LIN {X 0,Y 362.033,Z 639.51,A -85,B 0,C 180,E1 -13129.938,E2 -13129.938} C_VEL
LIN {X 0,Y 362.163,Z 639.495,A -85,B 0,C 180,E1 -13133.314,E2 -13133.314} C_VEL
LIN {X 0,Y 362.282,Z 639.48,A -85,B 0,C 180,E1 -13137.777,E2 -13137.777} C_VEL
LIN {X 0,Y 362.428,Z 639.459,A -85,B 0,C 180,E1 -13140,E2 -13140} C_VEL
LIN {X 0,Y 362.282,Z 639.48,A -85,B 0,C 180,E1 -13142.224,E2 -13142.224} C_VEL
LIN {X 0,Y 362.162,Z 639.494,A -85,B 0,C 180,E1 -13146.687,E2 -13146.687} C_VEL
LIN {X 0,Y 362.033,Z 639.507,A -85,B 0,C 180,E1 -13150.062,E2 -13150.062} C_VEL
LIN {X 0,Y 362,Z 639.515,A -85,B 0,C 180,E1 -13153.899,E2 -13153.899} C_VEL
LIN {X 0,Y 361.969,Z 639.52,A -85,B 0,C 180,E1 -13157.939,E2 -13157.939} C_VEL
LIN {X 0,Y 361.863,Z 639.533,A -85,B 0,C 180,E1 -13161.655,E2 -13161.655} C_VEL
LIN {X 0,Y 361.897,Z 639.53,A -85,B 0,C 180,E1 -13165.293,E2 -13165.293} C_VEL
LIN {X 0,Y 361.857,Z 639.512,A -85,B 0,C 180,E1 -13169.074,E2 -13169.074} C_VEL
LIN {X 0,Y 361.851,Z 639.537,A -85,B 0,C 180,E1 -13172.945,E2 -13172.945} C_VEL
LIN {X 0,Y 361.87,Z 639.533,A -85,B 0,C 180,E1 -13175.637,E2 -13175.637} C_VEL
LIN {X 0,Y 361.828,Z 639.538,A -85,B 0,C 180,E1 -13179.019,E2 -13179.019} C_VEL
LIN {X 0,Y 361.835,Z 639.538,A -85,B 0,C 180,E1 -13182.83,E2 -13182.83} C_VEL
LIN {X 0,Y 361.816,Z 639.535,A -85,B 0,C 180,E1 -13185.948,E2 -13185.948} C_VEL
LIN {X 0,Y 361.815,Z 639.547,A -85,B 0,C 180,E1 -13189.249,E2 -13189.249} C_VEL
LIN {X 0,Y 361.865,Z 639.536,A -85,B 0,C 180,E1 -13192.982,E2 -13192.982} C_VEL
LIN {X 0,Y 361.901,Z 639.566,A -85,B 0,C 180,E1 -13195.556,E2 -13195.556} C_VEL
LIN {X 0,Y 363.403,Z 645.852,A -85,B 0,C 180,E1 -13197.377,E2 -13197.377} C_VEL
LIN {X 0,Y 373.289,Z 667.329,A -85,B 0,C 180,E1 -13198.706,E2 -13198.706} C_VEL
LIN {X 0,Y 376.563,Z 675.649,A -85,B 0,C 180,E1 -13199.152,E2 -13199.152} C_VEL
LIN {X 0,Y 374.284,Z 781.835,A -85,B 0,C 180,E1 -13201.238,E2 -13201.238} C_VEL
LIN {X 0,Y 373.515,Z 795.857,A -85,B 0,C 180,E1 -13201.711,E2 -13201.711} C_VEL
LIN {X 0,Y 372.555,Z 809.132,A -85,B 0,C 180,E1 -13202.368,E2 -13202.368} C_VEL
LIN {X 0,Y 371.596,Z 819.142,A -85,B 0,C 180,E1 -13203.005,E2 -13203.005} C_VEL
LIN {X 0,Y 370.352,Z 831.212,A -85,B 0,C 180,E1 -13203.971,E2 -13203.971} C_VEL
LIN {X 0,Y 368.834,Z 843.683,A -85,B 0,C 180,E1 -13205.216,E2 -13205.216} C_VEL
LIN {X 0,Y 367.454,Z 854.256,A -85,B 0,C 180,E1 -13206.521,E2 -13206.521} C_VEL
LIN {X 0,Y 366.023,Z 864.257,A -85,B 0,C 180,E1 -13208.012,E2 -13208.012} C_VEL
LIN {X 0,Y 364.6,Z 873.584,A -85,B 0,C 180,E1 -13209.698,E2 -13209.698} C_VEL
LIN {X 0,Y 363.383,Z 881.912,A -85,B 0,C 180,E1 -13211.543,E2 -13211.543} C_VEL
LIN {X 0,Y 362.532,Z 887.72,A -85,B 0,C 180,E1 -13213.095,E2 -13213.095} C_VEL
LIN {X 0,Y 361.781,Z 892.985,A -85,B 0,C 180,E1 -13214.796,E2 -13214.796} C_VEL
LIN {X 0,Y 361.244,Z 897.486,A -85,B 0,C 180,E1 -13216.596,E2 -13216.596} C_VEL
LIN {X 0,Y 360.734,Z 901.59,A -85,B 0,C 180,E1 -13218.766,E2 -13218.766} C_VEL
LIN {X 0,Y 360.461,Z 904.443,A -85,B 0,C 180,E1 -13221.027,E2 -13221.027} C_VEL
LIN {X 0,Y 360.467,Z 905.926,A -85,B 0,C 180,E1 -13223.282,E2 -13223.282} C_VEL
LIN {X 0,Y 360.37,Z 906.095,A -85,B 0,C 180,E1 -13225.526,E2 -13225.526} C_VEL
LIN {X 0,Y 360.392,Z 904.952,A -85,B 0,C 180,E1 -13227.765,E2 -13227.765} C_VEL
LIN {X 0,Y 360.515,Z 902.485,A -85,B 0,C 180,E1 -13230,E2 -13230} C_VEL
LIN {X 0,Y 360.766,Z 898.613,A -85,B 0,C 180,E1 -13232.233,E2 -13232.233} C_VEL
LIN {X 0,Y 361.422,Z 893.189,A -85,B 0,C 180,E1 -13234.461,E2 -13234.461} C_VEL
LIN {X 0,Y 362.01,Z 888.061,A -85,B 0,C 180,E1 -13236.13,E2 -13236.13} C_VEL
LIN {X 0,Y 362.958,Z 880.664,A -85,B 0,C 180,E1 -13238.07,E2 -13238.07} C_VEL
LIN {X 0,Y 363.669,Z 872.986,A -85,B 0,C 180,E1 -13239.736,E2 -13239.736} C_VEL
LIN {X 0,Y 364.986,Z 863.701,A -85,B 0,C 180,E1 -13241.383,E2 -13241.383} C_VEL
LIN {X 0,Y 366.436,Z 852.377,A -85,B 0,C 180,E1 -13243.024,E2 -13243.024} C_VEL
LIN {X 0,Y 367.722,Z 840.85,A -85,B 0,C 180,E1 -13244.387,E2 -13244.387} C_VEL
LIN {X 0,Y 368.815,Z 829.618,A -85,B 0,C 180,E1 -13245.473,E2 -13245.473} C_VEL
LIN {X 0,Y 369.931,Z 817.471,A -85,B 0,C 180,E1 -13246.415,E2 -13246.415} C_VEL
LIN {X 0,Y 370.111,Z 815.428,A -85,B 0,C 180,E1 -13246.554,E2 -13246.554} C_VEL
LIN {X 0,Y 369.924,Z 810.057,A -85,B 0,C 180,E1 -13246.937,E2 -13246.937} C_VEL
LIN {X 0,Y 367.817,Z 801.278,A -85,B 0,C 180,E1 -13247.579,E2 -13247.579} C_VEL
LIN {X 0,Y 365.572,Z 792.287,A -85,B 0,C 180,E1 -13248.129,E2 -13248.129} C_VEL
LIN {X 0,Y 365.156,Z 786.588,A -85,B 0,C 180,E1 -13248.36,E2 -13248.36} C_VEL
LIN {X 0,Y 365.604,Z 770.654,A -85,B 0,C 180,E1 -13248.747,E2 -13248.747} C_VEL
LIN {X 0,Y 367.59,Z 676.095,A -85,B 0,C 180,E1 -13250.589,E2 -13250.589} C_VEL
LIN {X 0,Y 366.45,Z 671.797,A -85,B 0,C 180,E1 -13250.758,E2 -13250.758} C_VEL
LIN {X 0,Y 359.221,Z 653.429,A -85,B 0,C 180,E1 -13251.672,E2 -13251.672} C_VEL
LIN {X 0,Y 356.012,Z 645.71,A -85,B 0,C 180,E1 -13252.098,E2 -13252.098} C_VEL
LIN {X 0,Y 354.846,Z 640.411,A -85,B 0,C 180,E1 -13253.622,E2 -13253.622} C_VEL
LIN {X 0,Y 354.796,Z 640.417,A -85,B 0,C 180,E1 -13257.104,E2 -13257.104} C_VEL
LIN {X 0,Y 354.796,Z 640.415,A -85,B 0,C 180,E1 -13259.684,E2 -13259.684} C_VEL
LIN {X 0,Y 354.81,Z 640.412,A -85,B 0,C 180,E1 -13263.702,E2 -13263.702} C_VEL
LIN {X 0,Y 354.795,Z 640.414,A -85,B 0,C 180,E1 -13266.46,E2 -13266.46} C_VEL
LIN {X 0,Y 354.771,Z 640.403,A -85,B 0,C 180,E1 -13269.412,E2 -13269.412} C_VEL
LIN {X 0,Y 354.787,Z 640.418,A -85,B 0,C 180,E1 -13272.866,E2 -13272.866} C_VEL
LIN {X 0,Y 354.766,Z 640.416,A -85,B 0,C 180,E1 -13276.103,E2 -13276.103} C_VEL
LIN {X 0,Y 354.767,Z 640.42,A -85,B 0,C 180,E1 -13279.175,E2 -13279.175} C_VEL
LIN {X 0,Y 354.802,Z 640.391,A -85,B 0,C 180,E1 -13282.404,E2 -13282.404} C_VEL
LIN {X 0,Y 354.811,Z 640.403,A -85,B 0,C 180,E1 -13284.94,E2 -13284.94} C_VEL
LIN {X 0,Y 354.796,Z 640.41,A -85,B 0,C 180,E1 -13288.405,E2 -13288.405} C_VEL
LIN {X 0,Y 354.802,Z 640.415,A -85,B 0,C 180,E1 -13291.614,E2 -13291.614} C_VEL
LIN {X 0,Y 354.837,Z 640.397,A -85,B 0,C 180,E1 -13295.657,E2 -13295.657} C_VEL
LIN {X 0,Y 354.829,Z 640.41,A -85,B 0,C 180,E1 -13299.113,E2 -13299.113} C_VEL
LIN {X 0,Y 354.883,Z 640.386,A -85,B 0,C 180,E1 -13302.719,E2 -13302.719} C_VEL
LIN {X 0,Y 354.954,Z 640.393,A -85,B 0,C 180,E1 -13306.255,E2 -13306.255} C_VEL
LIN {X 0,Y 354.959,Z 640.38,A -85,B 0,C 180,E1 -13309.735,E2 -13309.735} C_VEL
LIN {X 0,Y 355.092,Z 640.377,A -85,B 0,C 180,E1 -13313.18,E2 -13313.18} C_VEL
LIN {X 0,Y 355.243,Z 640.36,A -85,B 0,C 180,E1 -13317.732,E2 -13317.732} C_VEL
LIN {X 0,Y 355.376,Z 640.338,A -85,B 0,C 180,E1 -13320,E2 -13320} C_VEL
LIN {X 0,Y 355.245,Z 640.358,A -85,B 0,C 180,E1 -13322.267,E2 -13322.267} C_VEL
LIN {X 0,Y 355.115,Z 640.37,A -85,B 0,C 180,E1 -13326.819,E2 -13326.819} C_VEL
LIN {X 0,Y 355.006,Z 640.386,A -85,B 0,C 180,E1 -13329.112,E2 -13329.112} C_VEL
LIN {X 0,Y 354.924,Z 640.397,A -85,B 0,C 180,E1 -13332.581,E2 -13332.581} C_VEL
LIN {X 0,Y 354.894,Z 640.398,A -85,B 0,C 180,E1 -13336.095,E2 -13336.095} C_VEL
LIN {X 0,Y 354.908,Z 640.396,A -85,B 0,C 180,E1 -13338.471,E2 -13338.471} C_VEL
LIN {X 0,Y 354.817,Z 640.413,A -85,B 0,C 180,E1 -13342.107,E2 -13342.107} C_VEL
LIN {X 0,Y 354.9,Z 640.4,A -85,B 0,C 180,E1 -13345.827,E2 -13345.827} C_VEL
LIN {X 0,Y 354.855,Z 640.406,A -85,B 0,C 180,E1 -13349.678,E2 -13349.678} C_VEL
LIN {X 0,Y 354.807,Z 640.411,A -85,B 0,C 180,E1 -13353.702,E2 -13353.702} C_VEL
LIN {X 0,Y 354.801,Z 640.414,A -85,B 0,C 180,E1 -13356.459,E2 -13356.459} C_VEL
LIN {X 0,Y 354.825,Z 640.406,A -85,B 0,C 180,E1 -13359.423,E2 -13359.423} C_VEL
LIN {X 0,Y 354.806,Z 640.413,A -85,B 0,C 180,E1 -13362.87,E2 -13362.87} C_VEL
LIN {X 0,Y 354.771,Z 640.414,A -85,B 0,C 180,E1 -13366.104,E2 -13366.104} C_VEL
LIN {X 0,Y 354.79,Z 640.415,A -85,B 0,C 180,E1 -13369.179,E2 -13369.179} C_VEL
LIN {X 0,Y 354.813,Z 640.415,A -85,B 0,C 180,E1 -13372.401,E2 -13372.401} C_VEL
LIN {X 0,Y 354.813,Z 640.415,A -85,B 0,C 180,E1 -13374.941,E2 -13374.941} C_VEL
LIN {X 0,Y 354.824,Z 640.498,A -85,B 0,C 180,E1 -13376.358,E2 -13376.358} C_VEL
LIN {X 0,Y 358.492,Z 655.954,A -85,B 0,C 180,E1 -13380.141,E2 -13380.141} C_VEL
LIN {X 0,Y 360.475,Z 665.739,A -85,B 0,C 180,E1 -13382.416,E2 -13382.416} C_VEL
LIN {X 0,Y 360.366,Z 669.663,A -85,B 0,C 180,E1 -13383.251,E2 -13383.251} C_VEL
LIN {X 0,Y 365.528,Z 699.808,A -85,B 0,C 180,E1 -13384.262,E2 -13384.262} C_VEL
LIN {X 0,Y 367.126,Z 709.941,A -85,B 0,C 180,E1 -13384.583,E2 -13384.583} C_VEL
LIN {X 0,Y 365.114,Z 807.088,A -85,B 0,C 180,E1 -13386.496,E2 -13386.496} C_VEL
LIN {X 0,Y 364.378,Z 821.425,A -85,B 0,C 180,E1 -13386.972,E2 -13386.972} C_VEL
LIN {X 0,Y 363.259,Z 835.788,A -85,B 0,C 180,E1 -13387.686,E2 -13387.686} C_VEL
LIN {X 0,Y 362.073,Z 848.948,A -85,B 0,C 180,E1 -13388.574,E2 -13388.574} C_VEL
LIN {X 0,Y 360.801,Z 861.127,A -85,B 0,C 180,E1 -13389.623,E2 -13389.623} C_VEL
LIN {X 0,Y 359.393,Z 872.902,A -85,B 0,C 180,E1 -13390.88,E2 -13390.88} C_VEL
LIN {X 0,Y 358.187,Z 881.703,A -85,B 0,C 180,E1 -13391.999,E2 -13391.999} C_VEL
LIN {X 0,Y 356.842,Z 892.714,A -85,B 0,C 180,E1 -13393.701,E2 -13393.701} C_VEL
LIN {X 0,Y 355.6,Z 902.545,A -85,B 0,C 180,E1 -13395.563,E2 -13395.563} C_VEL
LIN {X 0,Y 354.778,Z 910.501,A -85,B 0,C 180,E1 -13397.414,E2 -13397.414} C_VEL
LIN {X 0,Y 354.09,Z 916.591,A -85,B 0,C 180,E1 -13399.131,E2 -13399.131} C_VEL
LIN {X 0,Y 353.686,Z 921.635,A -85,B 0,C 180,E1 -13400.853,E2 -13400.853} C_VEL
LIN {X 0,Y 353.391,Z 926.828,A -85,B 0,C 180,E1 -13403.147,E2 -13403.147} C_VEL
LIN {X 0,Y 353.329,Z 928.844,A -85,B 0,C 180,E1 -13404.292,E2 -13404.292} C_VEL
LIN {X 0,Y 353.224,Z 931.786,A -85,B 0,C 180,E1 -13406.578,E2 -13406.578} C_VEL
LIN {X 0,Y 353.287,Z 933.347,A -85,B 0,C 180,E1 -13408.86,E2 -13408.86} C_VEL
LIN {X 0,Y 353.328,Z 933.621,A -85,B 0,C 180,E1 -13410,E2 -13410} C_VEL
LIN {X 0,Y 353.199,Z 933.155,A -85,B 0,C 180,E1 -13412.281,E2 -13412.281} C_VEL
LIN {X 0,Y 353.273,Z 931.354,A -85,B 0,C 180,E1 -13414.564,E2 -13414.564} C_VEL
LIN {X 0,Y 353.394,Z 928.176,A -85,B 0,C 180,E1 -13416.853,E2 -13416.853} C_VEL
LIN {X 0,Y 353.707,Z 923.514,A -85,B 0,C 180,E1 -13419.146,E2 -13419.146} C_VEL
LIN {X 0,Y 354.35,Z 917.212,A -85,B 0,C 180,E1 -13421.44,E2 -13421.44} C_VEL
LIN {X 0,Y 355.297,Z 910.221,A -85,B 0,C 180,E1 -13423.44,E2 -13423.44} C_VEL
LIN {X 0,Y 356.34,Z 902.934,A -85,B 0,C 180,E1 -13425.149,E2 -13425.149} C_VEL
LIN {X 0,Y 357.58,Z 894.193,A -85,B 0,C 180,E1 -13426.852,E2 -13426.852} C_VEL
LIN {X 0,Y 359.167,Z 883.624,A -85,B 0,C 180,E1 -13428.54,E2 -13428.54} C_VEL
LIN {X 0,Y 360.968,Z 871.814,A -85,B 0,C 180,E1 -13430.069,E2 -13430.069} C_VEL
LIN {X 0,Y 362.531,Z 860.236,A -85,B 0,C 180,E1 -13431.288,E2 -13431.288} C_VEL
LIN {X 0,Y 364.076,Z 846.936,A -85,B 0,C 180,E1 -13432.411,E2 -13432.411} C_VEL
LIN {X 0,Y 365.535,Z 833.217,A -85,B 0,C 180,E1 -13433.288,E2 -13433.288} C_VEL
LIN {X 0,Y 366.701,Z 819.616,A -85,B 0,C 180,E1 -13433.921,E2 -13433.921} C_VEL
LIN {X 0,Y 367.402,Z 805.854,A -85,B 0,C 180,E1 -13434.36,E2 -13434.36} C_VEL
LIN {X 0,Y 369.645,Z 710.085,A -85,B 0,C 180,E1 -13436.255,E2 -13436.255} C_VEL
LIN {X 0,Y 365.236,Z 685.41,A -85,B 0,C 180,E1 -13437.163,E2 -13437.163} C_VEL
LIN {X 0,Y 361.772,Z 669.821,A -85,B 0,C 180,E1 -13437.814,E2 -13437.814} C_VEL
LIN {X 0,Y 361.611,Z 669.008,A -85,B 0,C 180,E1 -13437.928,E2 -13437.928} C_VEL
LIN {X 0,Y 358.984,Z 656.804,A -85,B 0,C 180,E1 -13440.924,E2 -13440.924} C_VEL
LIN {X 0,Y 355.716,Z 643.633,A -85,B 0,C 180,E1 -13444.366,E2 -13444.366} C_VEL
LIN {X 0,Y 354.851,Z 640.398,A -85,B 0,C 180,E1 -13445.295,E2 -13445.295} C_VEL
LIN {X 0,Y 354.837,Z 640.411,A -85,B 0,C 180,E1 -13449.331,E2 -13449.331} C_VEL
LIN {X 0,Y 354.804,Z 640.411,A -85,B 0,C 180,E1 -13452.87,E2 -13452.87} C_VEL
LIN {X 0,Y 354.776,Z 640.416,A -85,B 0,C 180,E1 -13456.105,E2 -13456.105} C_VEL
LIN {X 0,Y 354.824,Z 640.405,A -85,B 0,C 180,E1 -13459.184,E2 -13459.184} C_VEL
LIN {X 0,Y 354.809,Z 640.395,A -85,B 0,C 180,E1 -13462.402,E2 -13462.402} C_VEL
LIN {X 0,Y 354.813,Z 640.41,A -85,B 0,C 180,E1 -13464.941,E2 -13464.941} C_VEL
LIN {X 0,Y 354.793,Z 640.389,A -85,B 0,C 180,E1 -13468.405,E2 -13468.405} C_VEL
LIN {X 0,Y 354.851,Z 640.407,A -85,B 0,C 180,E1 -13471.619,E2 -13471.619} C_VEL
LIN {X 0,Y 354.9,Z 640.397,A -85,B 0,C 180,E1 -13474.173,E2 -13474.173} C_VEL
LIN {X 0,Y 354.835,Z 640.404,A -85,B 0,C 180,E1 -13477.894,E2 -13477.894} C_VEL
LIN {X 0,Y 354.924,Z 640.392,A -85,B 0,C 180,E1 -13481.891,E2 -13481.891} C_VEL
LIN {X 0,Y 354.944,Z 640.39,A -85,B 0,C 180,E1 -13485.981,E2 -13485.981} C_VEL
LIN {X 0,Y 354.979,Z 640.391,A -85,B 0,C 180,E1 -13489.736,E2 -13489.736} C_VEL
LIN {X 0,Y 355.126,Z 640.372,A -85,B 0,C 180,E1 -13493.181,E2 -13493.181} C_VEL
LIN {X 0,Y 355.245,Z 640.357,A -85,B 0,C 180,E1 -13497.733,E2 -13497.733} C_VEL
LIN {X 0,Y 355.376,Z 640.337,A -85,B 0,C 180,E1 -13500,E2 -13500} C_VEL
LIN {X 0,Y 355.245,Z 640.357,A -85,B 0,C 180,E1 -13502.268,E2 -13502.268} C_VEL
LIN {X 0,Y 355.126,Z 640.373,A -85,B 0,C 180,E1 -13506.82,E2 -13506.82} C_VEL
LIN {X 0,Y 354.979,Z 640.385,A -85,B 0,C 180,E1 -13510.264,E2 -13510.264} C_VEL
LIN {X 0,Y 354.945,Z 640.394,A -85,B 0,C 180,E1 -13514.019,E2 -13514.019} C_VEL
LIN {X 0,Y 354.924,Z 640.398,A -85,B 0,C 180,E1 -13518.109,E2 -13518.109} C_VEL
LIN {X 0,Y 354.817,Z 640.411,A -85,B 0,C 180,E1 -13522.108,E2 -13522.108} C_VEL
LIN {X 0,Y 354.83,Z 640.409,A -85,B 0,C 180,E1 -13525.833,E2 -13525.833} C_VEL
LIN {X 0,Y 354.801,Z 640.392,A -85,B 0,C 180,E1 -13529.684,E2 -13529.684} C_VEL
LIN {X 0,Y 354.789,Z 640.415,A -85,B 0,C 180,E1 -13532.334,E2 -13532.334} C_VEL
LIN {X 0,Y 354.824,Z 640.41,A -85,B 0,C 180,E1 -13535.7,E2 -13535.7} C_VEL
LIN {X 0,Y 354.77,Z 640.412,A -85,B 0,C 180,E1 -13539.413,E2 -13539.413} C_VEL
LIN {X 0,Y 354.787,Z 640.417,A -85,B 0,C 180,E1 -13542.867,E2 -13542.867} C_VEL
LIN {X 0,Y 354.765,Z 640.414,A -85,B 0,C 180,E1 -13546.103,E2 -13546.103} C_VEL
LIN {X 0,Y 354.768,Z 640.425,A -85,B 0,C 180,E1 -13549.176,E2 -13549.176} C_VEL
LIN {X 0,Y 354.802,Z 640.416,A -85,B 0,C 180,E1 -13552.405,E2 -13552.405} C_VEL
LIN {X 0,Y 354.87,Z 640.462,A -85,B 0,C 180,E1 -13555.028,E2 -13555.028} C_VEL
LIN {X 0,Y 356.235,Z 646.109,A -85,B 0,C 180,E1 -13556.718,E2 -13556.718} C_VEL
LIN {X 0,Y 366.574,Z 668.221,A -85,B 0,C 180,E1 -13558.154,E2 -13558.154} C_VEL
LIN {X 0,Y 370.262,Z 677.295,A -85,B 0,C 180,E1 -13558.667,E2 -13558.667} C_VEL
LIN {X 0,Y 367.886,Z 782.415,A -85,B 0,C 180,E1 -13560.769,E2 -13560.769} C_VEL
LIN {X 0,Y 367.076,Z 797.106,A -85,B 0,C 180,E1 -13561.286,E2 -13561.286} C_VEL
LIN {X 0,Y 366.02,Z 810.282,A -85,B 0,C 180,E1 -13561.959,E2 -13561.959} C_VEL
LIN {X 0,Y 365.025,Z 820.541,A -85,B 0,C 180,E1 -13562.634,E2 -13562.634} C_VEL
LIN {X 0,Y 363.539,Z 833.851,A -85,B 0,C 180,E1 -13563.754,E2 -13563.754} C_VEL
LIN {X 0,Y 361.967,Z 845.818,A -85,B 0,C 180,E1 -13565.02,E2 -13565.02} C_VEL
LIN {X 0,Y 360.527,Z 856.284,A -85,B 0,C 180,E1 -13566.379,E2 -13566.379} C_VEL
LIN {X 0,Y 359.094,Z 865.815,A -85,B 0,C 180,E1 -13567.868,E2 -13567.868} C_VEL
LIN {X 0,Y 357.615,Z 874.918,A -85,B 0,C 180,E1 -13569.584,E2 -13569.584} C_VEL
LIN {X 0,Y 356.332,Z 883.589,A -85,B 0,C 180,E1 -13571.605,E2 -13571.605} C_VEL
LIN {X 0,Y 355.347,Z 889.653,A -85,B 0,C 180,E1 -13573.335,E2 -13573.335} C_VEL
LIN {X 0,Y 354.435,Z 896.073,A -85,B 0,C 180,E1 -13575.649,E2 -13575.649} C_VEL
LIN {X 0,Y 353.92,Z 899.781,A -85,B 0,C 180,E1 -13577.383,E2 -13577.383} C_VEL
LIN {X 0,Y 353.476,Z 903.387,A -85,B 0,C 180,E1 -13579.692,E2 -13579.692} C_VEL
LIN {X 0,Y 353.338,Z 905.583,A -85,B 0,C 180,E1 -13581.997,E2 -13581.997} C_VEL
LIN {X 0,Y 353.317,Z 906.405,A -85,B 0,C 180,E1 -13584.035,E2 -13584.035} C_VEL
LIN {X 0,Y 353.28,Z 906.377,A -85,B 0,C 180,E1 -13585.436,E2 -13585.436} C_VEL
LIN {X 0,Y 353.292,Z 905.269,A -85,B 0,C 180,E1 -13587.72,E2 -13587.72} C_VEL
LIN {X 0,Y 353.45,Z 902.837,A -85,B 0,C 180,E1 -13590,E2 -13590} C_VEL
LIN {X 0,Y 353.709,Z 899.017,A -85,B 0,C 180,E1 -13592.278,E2 -13592.278} C_VEL
LIN {X 0,Y 354.386,Z 893.638,A -85,B 0,C 180,E1 -13594.55,E2 -13594.55} C_VEL
LIN {X 0,Y 354.984,Z 888.539,A -85,B 0,C 180,E1 -13596.251,E2 -13596.251} C_VEL
LIN {X 0,Y 355.964,Z 881.204,A -85,B 0,C 180,E1 -13598.23,E2 -13598.23} C_VEL
LIN {X 0,Y 356.705,Z 873.739,A -85,B 0,C 180,E1 -13599.891,E2 -13599.891} C_VEL
LIN {X 0,Y 358.081,Z 864.354,A -85,B 0,C 180,E1 -13601.606,E2 -13601.606} C_VEL
LIN {X 0,Y 359.423,Z 854.174,A -85,B 0,C 180,E1 -13603.139,E2 -13603.139} C_VEL
LIN {X 0,Y 360.757,Z 842.962,A -85,B 0,C 180,E1 -13604.526,E2 -13604.526} C_VEL
LIN {X 0,Y 362.019,Z 830.579,A -85,B 0,C 180,E1 -13605.771,E2 -13605.771} C_VEL
LIN {X 0,Y 363.191,Z 818.604,A -85,B 0,C 180,E1 -13606.729,E2 -13606.729} C_VEL
LIN {X 0,Y 364.218,Z 805.46,A -85,B 0,C 180,E1 -13607.548,E2 -13607.548} C_VEL
LIN {X 0,Y 364.999,Z 791.191,A -85,B 0,C 180,E1 -13608.197,E2 -13608.197} C_VEL
LIN {X 0,Y 365.156,Z 786.588,A -85,B 0,C 180,E1 -13608.36,E2 -13608.36} C_VEL
LIN {X 0,Y 364.747,Z 780.831,A -85,B 0,C 180,E1 -13608.567,E2 -13608.567} C_VEL
LIN {X 0,Y 359.828,Z 762.18,A -85,B 0,C 180,E1 -13609.303,E2 -13609.303} C_VEL
LIN {X 0,Y 359.382,Z 756.37,A -85,B 0,C 180,E1 -13609.454,E2 -13609.454} C_VEL
LIN {X 0,Y 361.125,Z 677.298,A -85,B 0,C 180,E1 -13611.019,E2 -13611.019} C_VEL
LIN {X 0,Y 359.464,Z 672.117,A -85,B 0,C 180,E1 -13611.25,E2 -13611.25} C_VEL
LIN {X 0,Y 352.59,Z 654.789,A -85,B 0,C 180,E1 -13612.144,E2 -13612.144} C_VEL
LIN {X 0,Y 348.833,Z 645.917,A -85,B 0,C 180,E1 -13612.671,E2 -13612.671} C_VEL
LIN {X 0,Y 347.803,Z 641.288,A -85,B 0,C 180,E1 -13614.005,E2 -13614.005} C_VEL
LIN {X 0,Y 347.731,Z 641.298,A -85,B 0,C 180,E1 -13617.701,E2 -13617.701} C_VEL
LIN {X 0,Y 347.732,Z 641.297,A -85,B 0,C 180,E1 -13620.35,E2 -13620.35} C_VEL
LIN {X 0,Y 347.751,Z 641.292,A -85,B 0,C 180,E1 -13624.043,E2 -13624.043} C_VEL
LIN {X 0,Y 347.758,Z 641.292,A -85,B 0,C 180,E1 -13627.322,E2 -13627.322} C_VEL
LIN {X 0,Y 347.744,Z 641.292,A -85,B 0,C 180,E1 -13631.601,E2 -13631.601} C_VEL
LIN {X 0,Y 347.704,Z 641.299,A -85,B 0,C 180,E1 -13635.027,E2 -13635.027} C_VEL
LIN {X 0,Y 347.742,Z 641.291,A -85,B 0,C 180,E1 -13638.399,E2 -13638.399} C_VEL
LIN {X 0,Y 347.758,Z 641.266,A -85,B 0,C 180,E1 -13642.678,E2 -13642.678} C_VEL
LIN {X 0,Y 347.751,Z 641.29,A -85,B 0,C 180,E1 -13645.956,E2 -13645.956} C_VEL
LIN {X 0,Y 347.744,Z 641.282,A -85,B 0,C 180,E1 -13649.651,E2 -13649.651} C_VEL
LIN {X 0,Y 347.751,Z 641.29,A -85,B 0,C 180,E1 -13653.601,E2 -13653.601} C_VEL
LIN {X 0,Y 347.768,Z 641.277,A -85,B 0,C 180,E1 -13656.16,E2 -13656.16} C_VEL
LIN {X 0,Y 347.803,Z 641.283,A -85,B 0,C 180,E1 -13659.908,E2 -13659.908} C_VEL
LIN {X 0,Y 347.835,Z 641.27,A -85,B 0,C 180,E1 -13663.568,E2 -13663.568} C_VEL
LIN {X 0,Y 347.893,Z 641.274,A -85,B 0,C 180,E1 -13667.16,E2 -13667.16} C_VEL
LIN {X 0,Y 347.938,Z 641.257,A -85,B 0,C 180,E1 -13670.7,E2 -13670.7} C_VEL
LIN {X 0,Y 348.046,Z 641.252,A -85,B 0,C 180,E1 -13674.205,E2 -13674.205} C_VEL
LIN {X 0,Y 348.205,Z 641.236,A -85,B 0,C 180,E1 -13677.686,E2 -13677.686} C_VEL
LIN {X 0,Y 348.326,Z 641.216,A -85,B 0,C 180,E1 -13680,E2 -13680} C_VEL
LIN {X 0,Y 348.208,Z 641.234,A -85,B 0,C 180,E1 -13682.313,E2 -13682.313} C_VEL
LIN {X 0,Y 348.083,Z 641.246,A -85,B 0,C 180,E1 -13686.958,E2 -13686.958} C_VEL
LIN {X 0,Y 347.947,Z 641.266,A -85,B 0,C 180,E1 -13689.299,E2 -13689.299} C_VEL
LIN {X 0,Y 347.892,Z 641.272,A -85,B 0,C 180,E1 -13692.839,E2 -13692.839} C_VEL
LIN {X 0,Y 347.843,Z 641.279,A -85,B 0,C 180,E1 -13696.431,E2 -13696.431} C_VEL
LIN {X 0,Y 347.857,Z 641.272,A -85,B 0,C 180,E1 -13698.86,E2 -13698.86} C_VEL
LIN {X 0,Y 347.764,Z 641.286,A -85,B 0,C 180,E1 -13702.58,E2 -13702.58} C_VEL
LIN {X 0,Y 347.812,Z 641.281,A -85,B 0,C 180,E1 -13705.108,E2 -13705.108} C_VEL
LIN {X 0,Y 347.812,Z 641.278,A -85,B 0,C 180,E1 -13707.693,E2 -13707.693} C_VEL
LIN {X 0,Y 347.765,Z 641.289,A -85,B 0,C 180,E1 -13710.346,E2 -13710.346} C_VEL
LIN {X 0,Y 347.746,Z 641.292,A -85,B 0,C 180,E1 -13714.464,E2 -13714.464} C_VEL
LIN {X 0,Y 347.777,Z 641.289,A -85,B 0,C 180,E1 -13717.989,E2 -13717.989} C_VEL
LIN {X 0,Y 347.767,Z 641.288,A -85,B 0,C 180,E1 -13721.828,E2 -13721.828} C_VEL
LIN {X 0,Y 347.768,Z 641.289,A -85,B 0,C 180,E1 -13725.016,E2 -13725.016} C_VEL
LIN {X 0,Y 347.752,Z 641.293,A -85,B 0,C 180,E1 -13728.397,E2 -13728.397} C_VEL
LIN {X 0,Y 347.778,Z 641.289,A -85,B 0,C 180,E1 -13732.01,E2 -13732.01} C_VEL
LIN {X 0,Y 347.745,Z 641.295,A -85,B 0,C 180,E1 -13735.536,E2 -13735.536} C_VEL
LIN {X 0,Y 347.79,Z 641.514,A -85,B 0,C 180,E1 -13735.946,E2 -13735.946} C_VEL
LIN {X 0,Y 350.787,Z 654.007,A -85,B 0,C 180,E1 -13739.1,E2 -13739.1} C_VEL
LIN {X 0,Y 353.5,Z 666.713,A -85,B 0,C 180,E1 -13742.147,E2 -13742.147} C_VEL
LIN {X 0,Y 353.652,Z 669.514,A -85,B 0,C 180,E1 -13742.757,E2 -13742.757} C_VEL
LIN {X 0,Y 358.623,Z 698.233,A -85,B 0,C 180,E1 -13743.746,E2 -13743.746} C_VEL
LIN {X 0,Y 360.601,Z 711.118,A -85,B 0,C 180,E1 -13744.161,E2 -13744.161} C_VEL
LIN {X 0,Y 358.567,Z 805.211,A -85,B 0,C 180,E1 -13746.04,E2 -13746.04} C_VEL
LIN {X 0,Y 357.824,Z 819.341,A -85,B 0,C 180,E1 -13746.487,E2 -13746.487} C_VEL
LIN {X 0,Y 356.792,Z 833.767,A -85,B 0,C 180,E1 -13747.182,E2 -13747.182} C_VEL
LIN {X 0,Y 355.537,Z 847.129,A -85,B 0,C 180,E1 -13748.068,E2 -13748.068} C_VEL
LIN {X 0,Y 354.051,Z 860.472,A -85,B 0,C 180,E1 -13749.217,E2 -13749.217} C_VEL
LIN {X 0,Y 352.63,Z 872.318,A -85,B 0,C 180,E1 -13750.498,E2 -13750.498} C_VEL
LIN {X 0,Y 351.155,Z 883.147,A -85,B 0,C 180,E1 -13751.928,E2 -13751.928} C_VEL
LIN {X 0,Y 349.735,Z 893.871,A -85,B 0,C 180,E1 -13753.66,E2 -13753.66} C_VEL
LIN {X 0,Y 348.583,Z 902.757,A -85,B 0,C 180,E1 -13755.411,E2 -13755.411} C_VEL
LIN {X 0,Y 347.761,Z 910.079,A -85,B 0,C 180,E1 -13757.156,E2 -13757.156} C_VEL
LIN {X 0,Y 347.08,Z 916.2,A -85,B 0,C 180,E1 -13758.909,E2 -13758.909} C_VEL
LIN {X 0,Y 346.524,Z 922.713,A -85,B 0,C 180,E1 -13761.251,E2 -13761.251} C_VEL
LIN {X 0,Y 346.315,Z 926.486,A -85,B 0,C 180,E1 -13763.006,E2 -13763.006} C_VEL
LIN {X 0,Y 346.195,Z 930.173,A -85,B 0,C 180,E1 -13765.342,E2 -13765.342} C_VEL
LIN {X 0,Y 346.125,Z 932.436,A -85,B 0,C 180,E1 -13767.672,E2 -13767.672} C_VEL
LIN {X 0,Y 346.233,Z 933.342,A -85,B 0,C 180,E1 -13770,E2 -13770} C_VEL
LIN {X 0,Y 346.108,Z 932.896,A -85,B 0,C 180,E1 -13772.327,E2 -13772.327} C_VEL
LIN {X 0,Y 346.19,Z 931.116,A -85,B 0,C 180,E1 -13774.658,E2 -13774.658} C_VEL
LIN {X 0,Y 346.319,Z 927.958,A -85,B 0,C 180,E1 -13776.994,E2 -13776.994} C_VEL
LIN {X 0,Y 346.661,Z 923.328,A -85,B 0,C 180,E1 -13779.334,E2 -13779.334} C_VEL
LIN {X 0,Y 347.368,Z 917.054,A -85,B 0,C 180,E1 -13781.673,E2 -13781.673} C_VEL
LIN {X 0,Y 348.359,Z 910.09,A -85,B 0,C 180,E1 -13783.712,E2 -13783.712} C_VEL
LIN {X 0,Y 349.44,Z 902.835,A -85,B 0,C 180,E1 -13785.455,E2 -13785.455} C_VEL
LIN {X 0,Y 350.77,Z 894.13,A -85,B 0,C 180,E1 -13787.189,E2 -13787.189} C_VEL
LIN {X 0,Y 352.427,Z 883.606,A -85,B 0,C 180,E1 -13788.908,E2 -13788.908} C_VEL
LIN {X 0,Y 354.307,Z 871.849,A -85,B 0,C 180,E1 -13790.463,E2 -13790.463} C_VEL
LIN {X 0,Y 356.036,Z 859.28,A -85,B 0,C 180,E1 -13791.809,E2 -13791.809} C_VEL
LIN {X 0,Y 357.524,Z 847.129,A -85,B 0,C 180,E1 -13792.844,E2 -13792.844} C_VEL
LIN {X 0,Y 359.06,Z 833.602,A -85,B 0,C 180,E1 -13793.733,E2 -13793.733} C_VEL
LIN {X 0,Y 360.267,Z 820.297,A -85,B 0,C 180,E1 -13794.375,E2 -13794.375} C_VEL
LIN {X 0,Y 361.051,Z 805.678,A -85,B 0,C 180,E1 -13794.855,E2 -13794.855} C_VEL
LIN {X 0,Y 363.361,Z 710.983,A -85,B 0,C 180,E1 -13796.761,E2 -13796.761} C_VEL
LIN {X 0,Y 358.734,Z 685.235,A -85,B 0,C 180,E1 -13797.74,E2 -13797.74} C_VEL
LIN {X 0,Y 355.938,Z 672.663,A -85,B 0,C 180,E1 -13798.281,E2 -13798.281} C_VEL
LIN {X 0,Y 354.429,Z 668.948,A -85,B 0,C 180,E1 -13798.539,E2 -13798.539} C_VEL
LIN {X 0,Y 352.075,Z 658.15,A -85,B 0,C 180,E1 -13801.265,E2 -13801.265} C_VEL
LIN {X 0,Y 348.935,Z 645.394,A -85,B 0,C 180,E1 -13804.679,E2 -13804.679} C_VEL
LIN {X 0,Y 347.79,Z 641.28,A -85,B 0,C 180,E1 -13805.875,E2 -13805.875} C_VEL
LIN {X 0,Y 347.766,Z 641.289,A -85,B 0,C 180,E1 -13808.791,E2 -13808.791} C_VEL
LIN {X 0,Y 347.766,Z 641.292,A -85,B 0,C 180,E1 -13811.828,E2 -13811.828} C_VEL
LIN {X 0,Y 347.737,Z 641.289,A -85,B 0,C 180,E1 -13815.022,E2 -13815.022} C_VEL
LIN {X 0,Y 347.768,Z 641.279,A -85,B 0,C 180,E1 -13818.394,E2 -13818.394} C_VEL
LIN {X 0,Y 347.777,Z 641.273,A -85,B 0,C 180,E1 -13822.011,E2 -13822.011} C_VEL
LIN {X 0,Y 347.745,Z 641.295,A -85,B 0,C 180,E1 -13825.536,E2 -13825.536} C_VEL
LIN {X 0,Y 347.764,Z 641.27,A -85,B 0,C 180,E1 -13829.654,E2 -13829.654} C_VEL
LIN {X 0,Y 347.852,Z 641.275,A -85,B 0,C 180,E1 -13832.745,E2 -13832.745} C_VEL
LIN {X 0,Y 347.789,Z 641.285,A -85,B 0,C 180,E1 -13836.162,E2 -13836.162} C_VEL
LIN {X 0,Y 347.818,Z 641.286,A -85,B 0,C 180,E1 -13839.91,E2 -13839.91} C_VEL
LIN {X 0,Y 347.868,Z 641.273,A -85,B 0,C 180,E1 -13842.36,E2 -13842.36} C_VEL
LIN {X 0,Y 347.898,Z 641.268,A -85,B 0,C 180,E1 -13845.971,E2 -13845.971} C_VEL
LIN {X 0,Y 347.93,Z 641.269,A -85,B 0,C 180,E1 -13849.526,E2 -13849.526} C_VEL
LIN {X 0,Y 348.092,Z 641.248,A -85,B 0,C 180,E1 -13853.042,E2 -13853.042} C_VEL
LIN {X 0,Y 348.208,Z 641.233,A -85,B 0,C 180,E1 -13857.687,E2 -13857.687} C_VEL
LIN {X 0,Y 348.327,Z 641.215,A -85,B 0,C 180,E1 -13860,E2 -13860} C_VEL
LIN {X 0,Y 348.208,Z 641.234,A -85,B 0,C 180,E1 -13862.314,E2 -13862.314} C_VEL
LIN {X 0,Y 348.092,Z 641.249,A -85,B 0,C 180,E1 -13866.958,E2 -13866.958} C_VEL
LIN {X 0,Y 347.93,Z 641.262,A -85,B 0,C 180,E1 -13870.475,E2 -13870.475} C_VEL
LIN {X 0,Y 347.9,Z 641.271,A -85,B 0,C 180,E1 -13874.15,E2 -13874.15} C_VEL
LIN {X 0,Y 347.893,Z 641.275,A -85,B 0,C 180,E1 -13878.291,E2 -13878.291} C_VEL
LIN {X 0,Y 347.769,Z 641.289,A -85,B 0,C 180,E1 -13881.627,E2 -13881.627} C_VEL
LIN {X 0,Y 347.779,Z 641.291,A -85,B 0,C 180,E1 -13885.111,E2 -13885.111} C_VEL
LIN {X 0,Y 347.743,Z 641.28,A -85,B 0,C 180,E1 -13887.7,E2 -13887.7} C_VEL
LIN {X 0,Y 347.742,Z 641.277,A -85,B 0,C 180,E1 -13890.349,E2 -13890.349} C_VEL
LIN {X 0,Y 347.75,Z 641.286,A -85,B 0,C 180,E1 -13894.044,E2 -13894.044} C_VEL
LIN {X 0,Y 347.759,Z 641.29,A -85,B 0,C 180,E1 -13897.322,E2 -13897.322} C_VEL
LIN {X 0,Y 347.743,Z 641.282,A -85,B 0,C 180,E1 -13901.601,E2 -13901.601} C_VEL
LIN {X 0,Y 347.704,Z 641.29,A -85,B 0,C 180,E1 -13905.028,E2 -13905.028} C_VEL
LIN {X 0,Y 347.743,Z 641.295,A -85,B 0,C 180,E1 -13908.399,E2 -13908.399} C_VEL
LIN {X 0,Y 347.758,Z 641.293,A -85,B 0,C 180,E1 -13912.679,E2 -13912.679} C_VEL
LIN {X 0,Y 347.802,Z 641.418,A -85,B 0,C 180,E1 -13914.483,E2 -13914.483} C_VEL
LIN {X 0,Y 349.139,Z 646.606,A -85,B 0,C 180,E1 -13916.04,E2 -13916.04} C_VEL
LIN {X 0,Y 359.506,Z 668.427,A -85,B 0,C 180,E1 -13917.53,E2 -13917.53} C_VEL
LIN {X 0,Y 363.981,Z 679.086,A -85,B 0,C 180,E1 -13918.167,E2 -13918.167} C_VEL
LIN {X 0,Y 361.584,Z 781.76,A -85,B 0,C 180,E1 -13920.248,E2 -13920.248} C_VEL
LIN {X 0,Y 360.784,Z 796.05,A -85,B 0,C 180,E1 -13920.737,E2 -13920.737} C_VEL
LIN {X 0,Y 359.749,Z 809.186,A -85,B 0,C 180,E1 -13921.399,E2 -13921.399} C_VEL
LIN {X 0,Y 358.627,Z 819.954,A -85,B 0,C 180,E1 -13922.103,E2 -13922.103} C_VEL
LIN {X 0,Y 357.301,Z 831.968,A -85,B 0,C 180,E1 -13923.102,E2 -13923.102} C_VEL
LIN {X 0,Y 355.833,Z 843.105,A -85,B 0,C 180,E1 -13924.245,E2 -13924.245} C_VEL
LIN {X 0,Y 354.155,Z 854.715,A -85,B 0,C 180,E1 -13925.706,E2 -13925.706} C_VEL
LIN {X 0,Y 352.424,Z 865.734,A -85,B 0,C 180,E1 -13927.426,E2 -13927.426} C_VEL
LIN {X 0,Y 350.869,Z 874.896,A -85,B 0,C 180,E1 -13929.174,E2 -13929.174} C_VEL
LIN {X 0,Y 349.465,Z 883.619,A -85,B 0,C 180,E1 -13931.23,E2 -13931.23} C_VEL
LIN {X 0,Y 348.44,Z 889.729,A -85,B 0,C 180,E1 -13932.995,E2 -13932.995} C_VEL
LIN {X 0,Y 347.455,Z 896.191,A -85,B 0,C 180,E1 -13935.355,E2 -13935.355} C_VEL
LIN {X 0,Y 346.765,Z 900.999,A -85,B 0,C 180,E1 -13937.713,E2 -13937.713} C_VEL
LIN {X 0,Y 346.416,Z 903.583,A -85,B 0,C 180,E1 -13939.479,E2 -13939.479} C_VEL
LIN {X 0,Y 346.269,Z 905.813,A -85,B 0,C 180,E1 -13941.832,E2 -13941.832} C_VEL
LIN {X 0,Y 346.245,Z 906.687,A -85,B 0,C 180,E1 -13944.044,E2 -13944.044} C_VEL
LIN {X 0,Y 346.173,Z 906.287,A -85,B 0,C 180,E1 -13946.508,E2 -13946.508} C_VEL
LIN {X 0,Y 346.279,Z 904.555,A -85,B 0,C 180,E1 -13948.837,E2 -13948.837} C_VEL
LIN {X 0,Y 346.476,Z 901.48,A -85,B 0,C 180,E1 -13951.162,E2 -13951.162} C_VEL
LIN {X 0,Y 346.953,Z 896.956,A -85,B 0,C 180,E1 -13953.484,E2 -13953.484} C_VEL
LIN {X 0,Y 347.814,Z 890.792,A -85,B 0,C 180,E1 -13955.799,E2 -13955.799} C_VEL
LIN {X 0,Y 348.38,Z 885.055,A -85,B 0,C 180,E1 -13957.535,E2 -13957.535} C_VEL
LIN {X 0,Y 349.018,Z 880.538,A -85,B 0,C 180,E1 -13958.686,E2 -13958.686} C_VEL
LIN {X 0,Y 349.93,Z 872.718,A -85,B 0,C 180,E1 -13960.414,E2 -13960.414} C_VEL
LIN {X 0,Y 351.438,Z 863.254,A -85,B 0,C 180,E1 -13962.121,E2 -13962.121} C_VEL
LIN {X 0,Y 352.831,Z 852.792,A -85,B 0,C 180,E1 -13963.682,E2 -13963.682} C_VEL
LIN {X 0,Y 354.243,Z 841.234,A -85,B 0,C 180,E1 -13965.094,E2 -13965.094} C_VEL
LIN {X 0,Y 355.456,Z 829.959,A -85,B 0,C 180,E1 -13966.217,E2 -13966.217} C_VEL
LIN {X 0,Y 356.642,Z 817.762,A -85,B 0,C 180,E1 -13967.193,E2 -13967.193} C_VEL
LIN {X 0,Y 357.699,Z 804.274,A -85,B 0,C 180,E1 -13968.026,E2 -13968.026} C_VEL
LIN {X 0,Y 358.432,Z 790.326,A -85,B 0,C 180,E1 -13968.654,E2 -13968.654} C_VEL
LIN {X 0,Y 358.952,Z 775.704,A -85,B 0,C 180,E1 -13969.07,E2 -13969.07} C_VEL
LIN {X 0,Y 359.382,Z 756.37,A -85,B 0,C 180,E1 -13969.454,E2 -13969.454} C_VEL
LIN {X 0,Y 358.925,Z 750.555,A -85,B 0,C 180,E1 -13969.608,E2 -13969.608} C_VEL
LIN {X 0,Y 354.041,Z 731.861,A -85,B 0,C 180,E1 -13970.348,E2 -13970.348} C_VEL
LIN {X 0,Y 353.629,Z 726.045,A -85,B 0,C 180,E1 -13970.504,E2 -13970.504} C_VEL
LIN {X 0,Y 354.658,Z 678.298,A -85,B 0,C 180,E1 -13971.47,E2 -13971.47} C_VEL
LIN {X 0,Y 346.979,Z 658.552,A -85,B 0,C 180,E1 -13972.501,E2 -13972.501} C_VEL
LIN {X 0,Y 341.693,Z 646.317,A -85,B 0,C 180,E1 -13973.212,E2 -13973.212} C_VEL
LIN {X 0,Y 340.738,Z 642.169,A -85,B 0,C 180,E1 -13974.447,E2 -13974.447} C_VEL
LIN {X 0,Y 340.681,Z 642.173,A -85,B 0,C 180,E1 -13978.325,E2 -13978.325} C_VEL
LIN {X 0,Y 340.685,Z 642.174,A -85,B 0,C 180,E1 -13981.046,E2 -13981.046} C_VEL
LIN {X 0,Y 340.718,Z 642.169,A -85,B 0,C 180,E1 -13985.279,E2 -13985.279} C_VEL
LIN {X 0,Y 340.696,Z 642.17,A -85,B 0,C 180,E1 -13988.382,E2 -13988.382} C_VEL
LIN {X 0,Y 340.696,Z 642.169,A -85,B 0,C 180,E1 -13992.044,E2 -13992.044} C_VEL
LIN {X 0,Y 340.652,Z 642.175,A -85,B 0,C 180,E1 -13996.227,E2 -13996.227} C_VEL
LIN {X 0,Y 340.672,Z 642.174,A -85,B 0,C 180,E1 -13998.688,E2 -13998.688} C_VEL
LIN {X 0,Y 340.721,Z 642.148,A -85,B 0,C 180,E1 -14001.77,E2 -14001.77} C_VEL
LIN {X 0,Y 340.725,Z 642.166,A -85,B 0,C 180,E1 -14005.595,E2 -14005.595} C_VEL
LIN {X 0,Y 340.697,Z 642.164,A -85,B 0,C 180,E1 -14008.955,E2 -14008.955} C_VEL
LIN {X 0,Y 340.722,Z 642.169,A -85,B 0,C 180,E1 -14013.012,E2 -14013.012} C_VEL
LIN {X 0,Y 340.743,Z 642.152,A -85,B 0,C 180,E1 -14015.637,E2 -14015.637} C_VEL
LIN {X 0,Y 340.733,Z 642.168,A -85,B 0,C 180,E1 -14019.473,E2 -14019.473} C_VEL
LIN {X 0,Y 340.795,Z 642.142,A -85,B 0,C 180,E1 -14021.98,E2 -14021.98} C_VEL
LIN {X 0,Y 340.872,Z 642.151,A -85,B 0,C 180,E1 -14025.705,E2 -14025.705} C_VEL
LIN {X 0,Y 340.851,Z 642.137,A -85,B 0,C 180,E1 -14029.305,E2 -14029.305} C_VEL
LIN {X 0,Y 341.005,Z 642.13,A -85,B 0,C 180,E1 -14032.896,E2 -14032.896} C_VEL
LIN {X 0,Y 340.833,Z 642.151,A -85,B 0,C 180,E1 -14035.268,E2 -14035.268} C_VEL
LIN {X 0,Y 341.167,Z 642.112,A -85,B 0,C 180,E1 -14037.638,E2 -14037.638} C_VEL
LIN {X 0,Y 341.277,Z 642.093,A -85,B 0,C 180,E1 -14040,E2 -14040} C_VEL
LIN {X 0,Y 341.17,Z 642.111,A -85,B 0,C 180,E1 -14042.361,E2 -14042.361} C_VEL
LIN {X 0,Y 341.053,Z 642.122,A -85,B 0,C 180,E1 -14047.102,E2 -14047.102} C_VEL
LIN {X 0,Y 340.873,Z 642.14,A -85,B 0,C 180,E1 -14050.693,E2 -14050.693} C_VEL
LIN {X 0,Y 340.865,Z 642.145,A -85,B 0,C 180,E1 -14054.324,E2 -14054.324} C_VEL
LIN {X 0,Y 340.84,Z 642.148,A -85,B 0,C 180,E1 -14058.467,E2 -14058.467} C_VEL
LIN {X 0,Y 340.719,Z 642.167,A -85,B 0,C 180,E1 -14061.841,E2 -14061.841} C_VEL
LIN {X 0,Y 340.773,Z 642.159,A -85,B 0,C 180,E1 -14065.664,E2 -14065.664} C_VEL
LIN {X 0,Y 340.742,Z 642.163,A -85,B 0,C 180,E1 -14068.319,E2 -14068.319} C_VEL
LIN {X 0,Y 340.706,Z 642.166,A -85,B 0,C 180,E1 -14071.044,E2 -14071.044} C_VEL
LIN {X 0,Y 340.72,Z 642.167,A -85,B 0,C 180,E1 -14075.278,E2 -14075.278} C_VEL
LIN {X 0,Y 340.719,Z 642.171,A -85,B 0,C 180,E1 -14078.388,E2 -14078.388} C_VEL
LIN {X 0,Y 340.734,Z 642.164,A -85,B 0,C 180,E1 -14082.052,E2 -14082.052} C_VEL
LIN {X 0,Y 340.685,Z 642.17,A -85,B 0,C 180,E1 -14085.461,E2 -14085.461} C_VEL
LIN {X 0,Y 340.687,Z 642.173,A -85,B 0,C 180,E1 -14088.69,E2 -14088.69} C_VEL
LIN {X 0,Y 340.736,Z 642.166,A -85,B 0,C 180,E1 -14091.773,E2 -14091.773} C_VEL
LIN {X 0,Y 340.715,Z 642.297,A -85,B 0,C 180,E1 -14095.458,E2 -14095.458} C_VEL
LIN {X 0,Y 343.608,Z 654.258,A -85,B 0,C 180,E1 -14098.563,E2 -14098.563} C_VEL
LIN {X 0,Y 346.226,Z 666.189,A -85,B 0,C 180,E1 -14101.512,E2 -14101.512} C_VEL
LIN {X 0,Y 346.708,Z 669.139,A -85,B 0,C 180,E1 -14102.21,E2 -14102.21} C_VEL
LIN {X 0,Y 349.029,Z 680.228,A -85,B 0,C 180,E1 -14102.641,E2 -14102.641} C_VEL
LIN {X 0,Y 354.088,Z 711.421,A -85,B 0,C 180,E1 -14103.705,E2 -14103.705} C_VEL
LIN {X 0,Y 352.057,Z 803.315,A -85,B 0,C 180,E1 -14105.568,E2 -14105.568} C_VEL
LIN {X 0,Y 351.304,Z 818.084,A -85,B 0,C 180,E1 -14106.023,E2 -14106.023} C_VEL
LIN {X 0,Y 350.29,Z 831.504,A -85,B 0,C 180,E1 -14106.656,E2 -14106.656} C_VEL
LIN {X 0,Y 349.069,Z 844.74,A -85,B 0,C 180,E1 -14107.509,E2 -14107.509} C_VEL
LIN {X 0,Y 347.574,Z 858.376,A -85,B 0,C 180,E1 -14108.656,E2 -14108.656} C_VEL
LIN {X 0,Y 346.042,Z 870.545,A -85,B 0,C 180,E1 -14109.957,E2 -14109.957} C_VEL
LIN {X 0,Y 344.598,Z 880.637,A -85,B 0,C 180,E1 -14111.263,E2 -14111.263} C_VEL
LIN {X 0,Y 343.096,Z 891.734,A -85,B 0,C 180,E1 -14113.028,E2 -14113.028} C_VEL
LIN {X 0,Y 341.864,Z 900.769,A -85,B 0,C 180,E1 -14114.776,E2 -14114.776} C_VEL
LIN {X 0,Y 340.938,Z 908.528,A -85,B 0,C 180,E1 -14116.591,E2 -14116.591} C_VEL
LIN {X 0,Y 340.056,Z 915.807,A -85,B 0,C 180,E1 -14118.677,E2 -14118.677} C_VEL
LIN {X 0,Y 339.473,Z 922.346,A -85,B 0,C 180,E1 -14121.067,E2 -14121.067} C_VEL
LIN {X 0,Y 339.198,Z 927.223,A -85,B 0,C 180,E1 -14123.456,E2 -14123.456} C_VEL
LIN {X 0,Y 339.097,Z 929.852,A -85,B 0,C 180,E1 -14125.244,E2 -14125.244} C_VEL
LIN {X 0,Y 339.036,Z 932.138,A -85,B 0,C 180,E1 -14127.624,E2 -14127.624} C_VEL
LIN {X 0,Y 339.138,Z 933.064,A -85,B 0,C 180,E1 -14130,E2 -14130} C_VEL
LIN {X 0,Y 339.02,Z 932.639,A -85,B 0,C 180,E1 -14132.376,E2 -14132.376} C_VEL
LIN {X 0,Y 339.093,Z 930.878,A -85,B 0,C 180,E1 -14134.755,E2 -14134.755} C_VEL
LIN {X 0,Y 339.245,Z 927.741,A -85,B 0,C 180,E1 -14137.14,E2 -14137.14} C_VEL
LIN {X 0,Y 339.628,Z 923.142,A -85,B 0,C 180,E1 -14139.529,E2 -14139.529} C_VEL
LIN {X 0,Y 340.393,Z 916.898,A -85,B 0,C 180,E1 -14141.915,E2 -14141.915} C_VEL
LIN {X 0,Y 341.442,Z 909.962,A -85,B 0,C 180,E1 -14143.996,E2 -14143.996} C_VEL
LIN {X 0,Y 342.535,Z 902.738,A -85,B 0,C 180,E1 -14145.775,E2 -14145.775} C_VEL
LIN {X 0,Y 343.968,Z 894.071,A -85,B 0,C 180,E1 -14147.54,E2 -14147.54} C_VEL
LIN {X 0,Y 345.687,Z 883.591,A -85,B 0,C 180,E1 -14149.291,E2 -14149.291} C_VEL
LIN {X 0,Y 347.66,Z 871.888,A -85,B 0,C 180,E1 -14150.873,E2 -14150.873} C_VEL
LIN {X 0,Y 349.26,Z 860.904,A -85,B 0,C 180,E1 -14152.088,E2 -14152.088} C_VEL
LIN {X 0,Y 350.797,Z 849.088,A -85,B 0,C 180,E1 -14153.152,E2 -14153.152} C_VEL
LIN {X 0,Y 352.336,Z 836.198,A -85,B 0,C 180,E1 -14154.058,E2 -14154.058} C_VEL
LIN {X 0,Y 353.659,Z 822.403,A -85,B 0,C 180,E1 -14154.783,E2 -14154.783} C_VEL
LIN {X 0,Y 354.609,Z 808.113,A -85,B 0,C 180,E1 -14155.299,E2 -14155.299} C_VEL
LIN {X 0,Y 356.222,Z 752.31,A -85,B 0,C 180,E1 -14156.454,E2 -14156.454} C_VEL
LIN {X 0,Y 357.09,Z 711.782,A -85,B 0,C 180,E1 -14157.289,E2 -14157.289} C_VEL
LIN {X 0,Y 352.445,Z 686.101,A -85,B 0,C 180,E1 -14158.298,E2 -14158.298} C_VEL
LIN {X 0,Y 350.187,Z 675.675,A -85,B 0,C 180,E1 -14158.755,E2 -14158.755} C_VEL
LIN {X 0,Y 347.222,Z 668.684,A -85,B 0,C 180,E1 -14159.229,E2 -14159.229} C_VEL
LIN {X 0,Y 344.816,Z 658.078,A -85,B 0,C 180,E1 -14162.001,E2 -14162.001} C_VEL
LIN {X 0,Y 341.983,Z 646.745,A -85,B 0,C 180,E1 -14165.129,E2 -14165.129} C_VEL
LIN {X 0,Y 340.71,Z 642.167,A -85,B 0,C 180,E1 -14166.486,E2 -14166.486} C_VEL
LIN {X 0,Y 340.709,Z 642.165,A -85,B 0,C 180,E1 -14169.751,E2 -14169.751} C_VEL
LIN {X 0,Y 340.711,Z 642.165,A -85,B 0,C 180,E1 -14172.899,E2 -14172.899} C_VEL
LIN {X 0,Y 340.711,Z 642.159,A -85,B 0,C 180,E1 -14177.101,E2 -14177.101} C_VEL
LIN {X 0,Y 340.71,Z 642.169,A -85,B 0,C 180,E1 -14180.249,E2 -14180.249} C_VEL
LIN {X 0,Y 340.711,Z 642.154,A -85,B 0,C 180,E1 -14183.559,E2 -14183.559} C_VEL
LIN {X 0,Y 340.694,Z 642.168,A -85,B 0,C 180,E1 -14186.154,E2 -14186.154} C_VEL
LIN {X 0,Y 340.775,Z 642.151,A -85,B 0,C 180,E1 -14190.333,E2 -14190.333} C_VEL
LIN {X 0,Y 340.805,Z 642.153,A -85,B 0,C 180,E1 -14193.02,E2 -14193.02} C_VEL
LIN {X 0,Y 340.729,Z 642.161,A -85,B 0,C 180,E1 -14196.927,E2 -14196.927} C_VEL
LIN {X 0,Y 340.796,Z 642.154,A -85,B 0,C 180,E1 -14200.734,E2 -14200.734} C_VEL
LIN {X 0,Y 340.789,Z 642.156,A -85,B 0,C 180,E1 -14203.219,E2 -14203.219} C_VEL
LIN {X 0,Y 340.845,Z 642.147,A -85,B 0,C 180,E1 -14206.891,E2 -14206.891} C_VEL
LIN {X 0,Y 340.915,Z 642.134,A -85,B 0,C 180,E1 -14210.508,E2 -14210.508} C_VEL
LIN {X 0,Y 341.06,Z 642.125,A -85,B 0,C 180,E1 -14212.898,E2 -14212.898} C_VEL
LIN {X 0,Y 341.169,Z 642.11,A -85,B 0,C 180,E1 -14217.639,E2 -14217.639} C_VEL
LIN {X 0,Y 341.277,Z 642.093,A -85,B 0,C 180,E1 -14220,E2 -14220} C_VEL
LIN {X 0,Y 341.169,Z 642.111,A -85,B 0,C 180,E1 -14222.362,E2 -14222.362} C_VEL
LIN {X 0,Y 341.06,Z 642.125,A -85,B 0,C 180,E1 -14227.102,E2 -14227.102} C_VEL
LIN {X 0,Y 340.872,Z 642.142,A -85,B 0,C 180,E1 -14230.694,E2 -14230.694} C_VEL
LIN {X 0,Y 340.865,Z 642.146,A -85,B 0,C 180,E1 -14234.325,E2 -14234.325} C_VEL
LIN {X 0,Y 340.839,Z 642.151,A -85,B 0,C 180,E1 -14238.467,E2 -14238.467} C_VEL
LIN {X 0,Y 340.719,Z 642.167,A -85,B 0,C 180,E1 -14241.842,E2 -14241.842} C_VEL
LIN {X 0,Y 340.754,Z 642.163,A -85,B 0,C 180,E1 -14244.839,E2 -14244.839} C_VEL
LIN {X 0,Y 340.687,Z 642.15,A -85,B 0,C 180,E1 -14248.325,E2 -14248.325} C_VEL
LIN {X 0,Y 340.696,Z 642.162,A -85,B 0,C 180,E1 -14251.045,E2 -14251.045} C_VEL
LIN {X 0,Y 340.72,Z 642.17,A -85,B 0,C 180,E1 -14255.279,E2 -14255.279} C_VEL
LIN {X 0,Y 340.696,Z 642.171,A -85,B 0,C 180,E1 -14258.383,E2 -14258.383} C_VEL
LIN {X 0,Y 340.695,Z 642.165,A -85,B 0,C 180,E1 -14262.045,E2 -14262.045} C_VEL
LIN {X 0,Y 340.652,Z 642.172,A -85,B 0,C 180,E1 -14266.228,E2 -14266.228} C_VEL
LIN {X 0,Y 340.673,Z 642.177,A -85,B 0,C 180,E1 -14268.689,E2 -14268.689} C_VEL
LIN {X 0,Y 340.721,Z 642.171,A -85,B 0,C 180,E1 -14271.771,E2 -14271.771} C_VEL
LIN {X 0,Y 340.751,Z 642.296,A -85,B 0,C 180,E1 -14273.89,E2 -14273.89} C_VEL
LIN {X 0,Y 341.915,Z 646.786,A -85,B 0,C 180,E1 -14275.306,E2 -14275.306} C_VEL
LIN {X 0,Y 353.037,Z 669.763,A -85,B 0,C 180,E1 -14276.959,E2 -14276.959} C_VEL
LIN {X 0,Y 357.728,Z 680.914,A -85,B 0,C 180,E1 -14277.65,E2 -14277.65} C_VEL
LIN {X 0,Y 355.259,Z 782.434,A -85,B 0,C 180,E1 -14279.746,E2 -14279.746} C_VEL
LIN {X 0,Y 354.417,Z 796.545,A -85,B 0,C 180,E1 -14280.24,E2 -14280.24} C_VEL
LIN {X 0,Y 353.261,Z 810.503,A -85,B 0,C 180,E1 -14280.968,E2 -14280.968} C_VEL
LIN {X 0,Y 352.106,Z 821.351,A -85,B 0,C 180,E1 -14281.703,E2 -14281.703} C_VEL
LIN {X 0,Y 350.509,Z 834.597,A -85,B 0,C 180,E1 -14282.861,E2 -14282.861} C_VEL
LIN {X 0,Y 348.988,Z 845.345,A -85,B 0,C 180,E1 -14284.023,E2 -14284.023} C_VEL
LIN {X 0,Y 347.359,Z 856.076,A -85,B 0,C 180,E1 -14285.44,E2 -14285.44} C_VEL
LIN {X 0,Y 345.79,Z 865.655,A -85,B 0,C 180,E1 -14286.968,E2 -14286.968} C_VEL
LIN {X 0,Y 344.155,Z 874.877,A -85,B 0,C 180,E1 -14288.748,E2 -14288.748} C_VEL
LIN {X 0,Y 342.775,Z 882.717,A -85,B 0,C 180,E1 -14290.589,E2 -14290.589} C_VEL
LIN {X 0,Y 341.569,Z 889.807,A -85,B 0,C 180,E1 -14292.642,E2 -14292.642} C_VEL
LIN {X 0,Y 340.495,Z 896.312,A -85,B 0,C 180,E1 -14295.048,E2 -14295.048} C_VEL
LIN {X 0,Y 339.928,Z 900.098,A -85,B 0,C 180,E1 -14296.855,E2 -14296.855} C_VEL
LIN {X 0,Y 339.361,Z 903.779,A -85,B 0,C 180,E1 -14299.258,E2 -14299.258} C_VEL
LIN {X 0,Y 339.188,Z 906.044,A -85,B 0,C 180,E1 -14301.66,E2 -14301.66} C_VEL
LIN {X 0,Y 339.138,Z 906.969,A -85,B 0,C 180,E1 -14304.053,E2 -14304.053} C_VEL
LIN {X 0,Y 339.096,Z 906.585,A -85,B 0,C 180,E1 -14306.435,E2 -14306.435} C_VEL
LIN {X 0,Y 339.181,Z 904.889,A -85,B 0,C 180,E1 -14308.813,E2 -14308.813} C_VEL
LIN {X 0,Y 339.398,Z 901.849,A -85,B 0,C 180,E1 -14311.187,E2 -14311.187} C_VEL
LIN {X 0,Y 339.89,Z 897.374,A -85,B 0,C 180,E1 -14313.557,E2 -14313.557} C_VEL
LIN {X 0,Y 340.773,Z 891.259,A -85,B 0,C 180,E1 -14315.919,E2 -14315.919} C_VEL
LIN {X 0,Y 341.371,Z 885.559,A -85,B 0,C 180,E1 -14317.69,E2 -14317.69} C_VEL
LIN {X 0,Y 342.015,Z 881.076,A -85,B 0,C 180,E1 -14318.866,E2 -14318.866} C_VEL
LIN {X 0,Y 342.974,Z 873.31,A -85,B 0,C 180,E1 -14320.628,E2 -14320.628} C_VEL
LIN {X 0,Y 344.526,Z 863.91,A -85,B 0,C 180,E1 -14322.368,E2 -14322.368} C_VEL
LIN {X 0,Y 345.992,Z 853.521,A -85,B 0,C 180,E1 -14323.958,E2 -14323.958} C_VEL
LIN {X 0,Y 347.458,Z 842.056,A -85,B 0,C 180,E1 -14325.396,E2 -14325.396} C_VEL
LIN {X 0,Y 348.691,Z 830.907,A -85,B 0,C 180,E1 -14326.541,E2 -14326.541} C_VEL
LIN {X 0,Y 349.919,Z 818.881,A -85,B 0,C 180,E1 -14327.534,E2 -14327.534} C_VEL
LIN {X 0,Y 351.017,Z 805.653,A -85,B 0,C 180,E1 -14328.382,E2 -14328.382} C_VEL
LIN {X 0,Y 351.836,Z 792.14,A -85,B 0,C 180,E1 -14329.017,E2 -14329.017} C_VEL
LIN {X 0,Y 352.355,Z 778.522,A -85,B 0,C 180,E1 -14329.442,E2 -14329.442} C_VEL
LIN {X 0,Y 353.629,Z 726.045,A -85,B 0,C 180,E1 -14330.504,E2 -14330.504} C_VEL
LIN {X 0,Y 353.22,Z 720.237,A -85,B 0,C 180,E1 -14330.66,E2 -14330.66} C_VEL
LIN {X 0,Y 348.351,Z 701.58,A -85,B 0,C 180,E1 -14331.431,E2 -14331.431} C_VEL
LIN {X 0,Y 347.855,Z 695.773,A -85,B 0,C 180,E1 -14331.598,E2 -14331.598} C_VEL
LIN {X 0,Y 348.121,Z 679.783,A -85,B 0,C 180,E1 -14331.934,E2 -14331.934} C_VEL
LIN {X 0,Y 340.985,Z 661.523,A -85,B 0,C 180,E1 -14332.92,E2 -14332.92} C_VEL
LIN {X 0,Y 334.498,Z 646.485,A -85,B 0,C 180,E1 -14333.858,E2 -14333.858} C_VEL
LIN {X 0,Y 333.684,Z 643.048,A -85,B 0,C 180,E1 -14334.913,E2 -14334.913} C_VEL
LIN {X 0,Y 333.648,Z 643.052,A -85,B 0,C 180,E1 -14337.785,E2 -14337.785} C_VEL
LIN {X 0,Y 333.657,Z 643.051,A -85,B 0,C 180,E1 -14340.366,E2 -14340.366} C_VEL
LIN {X 0,Y 333.638,Z 643.053,A -85,B 0,C 180,E1 -14343.209,E2 -14343.209} C_VEL
LIN {X 0,Y 333.676,Z 643.045,A -85,B 0,C 180,E1 -14346.139,E2 -14346.139} C_VEL
LIN {X 0,Y 333.605,Z 643.041,A -85,B 0,C 180,E1 -14349.199,E2 -14349.199} C_VEL
LIN {X 0,Y 333.631,Z 643.051,A -85,B 0,C 180,E1 -14352.499,E2 -14352.499} C_VEL
LIN {X 0,Y 333.596,Z 643.054,A -85,B 0,C 180,E1 -14355.954,E2 -14355.954} C_VEL
LIN {X 0,Y 333.605,Z 643.054,A -85,B 0,C 180,E1 -14359.324,E2 -14359.324} C_VEL
LIN {X 0,Y 333.664,Z 643.021,A -85,B 0,C 180,E1 -14363.168,E2 -14363.168} C_VEL
LIN {X 0,Y 333.675,Z 643.039,A -85,B 0,C 180,E1 -14365.341,E2 -14365.341} C_VEL
LIN {X 0,Y 333.632,Z 643.047,A -85,B 0,C 180,E1 -14368.222,E2 -14368.222} C_VEL
LIN {X 0,Y 333.657,Z 643.04,A -85,B 0,C 180,E1 -14371.022,E2 -14371.022} C_VEL
LIN {X 0,Y 333.698,Z 643.033,A -85,B 0,C 180,E1 -14375.088,E2 -14375.088} C_VEL
LIN {X 0,Y 333.667,Z 643.046,A -85,B 0,C 180,E1 -14379.018,E2 -14379.018} C_VEL
LIN {X 0,Y 333.743,Z 643.023,A -85,B 0,C 180,E1 -14381.586,E2 -14381.586} C_VEL
LIN {X 0,Y 333.811,Z 643.03,A -85,B 0,C 180,E1 -14385.576,E2 -14385.576} C_VEL
LIN {X 0,Y 333.82,Z 643.014,A -85,B 0,C 180,E1 -14389.077,E2 -14389.077} C_VEL
LIN {X 0,Y 333.96,Z 643.008,A -85,B 0,C 180,E1 -14392.746,E2 -14392.746} C_VEL
LIN {X 0,Y 333.797,Z 643.027,A -85,B 0,C 180,E1 -14395.169,E2 -14395.169} C_VEL
LIN {X 0,Y 334.104,Z 642.991,A -85,B 0,C 180,E1 -14397.588,E2 -14397.588} C_VEL
LIN {X 0,Y 334.228,Z 642.971,A -85,B 0,C 180,E1 -14400,E2 -14400} C_VEL
LIN {X 0,Y 334.107,Z 642.991,A -85,B 0,C 180,E1 -14402.411,E2 -14402.411} C_VEL
LIN {X 0,Y 334.009,Z 642.999,A -85,B 0,C 180,E1 -14406.039,E2 -14406.039} C_VEL
LIN {X 0,Y 333.972,Z 643.008,A -85,B 0,C 180,E1 -14408.484,E2 -14408.484} C_VEL
LIN {X 0,Y 333.794,Z 643.03,A -85,B 0,C 180,E1 -14412.154,E2 -14412.154} C_VEL
LIN {X 0,Y 333.781,Z 643.026,A -85,B 0,C 180,E1 -14415.886,E2 -14415.886} C_VEL
LIN {X 0,Y 333.799,Z 643.024,A -85,B 0,C 180,E1 -14418.655,E2 -14418.655} C_VEL
LIN {X 0,Y 333.658,Z 643.046,A -85,B 0,C 180,E1 -14422.28,E2 -14422.28} C_VEL
LIN {X 0,Y 333.737,Z 643.037,A -85,B 0,C 180,E1 -14426.246,E2 -14426.246} C_VEL
LIN {X 0,Y 333.712,Z 643.039,A -85,B 0,C 180,E1 -14428.972,E2 -14428.972} C_VEL
LIN {X 0,Y 333.648,Z 643.05,A -85,B 0,C 180,E1 -14432.588,E2 -14432.588} C_VEL
LIN {X 0,Y 333.678,Z 643.047,A -85,B 0,C 180,E1 -14436.138,E2 -14436.138} C_VEL
LIN {X 0,Y 333.673,Z 643.042,A -85,B 0,C 180,E1 -14439.188,E2 -14439.188} C_VEL
LIN {X 0,Y 333.676,Z 643.046,A -85,B 0,C 180,E1 -14442.508,E2 -14442.508} C_VEL
LIN {X 0,Y 333.622,Z 643.048,A -85,B 0,C 180,E1 -14445.959,E2 -14445.959} C_VEL
LIN {X 0,Y 333.648,Z 643.049,A -85,B 0,C 180,E1 -14449.315,E2 -14449.315} C_VEL
LIN {X 0,Y 333.668,Z 643.048,A -85,B 0,C 180,E1 -14453.167,E2 -14453.167} C_VEL
LIN {X 0,Y 333.695,Z 643.171,A -85,B 0,C 180,E1 -14454.973,E2 -14454.973} C_VEL
LIN {X 0,Y 336.57,Z 655.203,A -85,B 0,C 180,E1 -14458.18,E2 -14458.18} C_VEL
LIN {X 0,Y 339.544,Z 668.773,A -85,B 0,C 180,E1 -14461.607,E2 -14461.607} C_VEL
LIN {X 0,Y 341.322,Z 674.558,A -85,B 0,C 180,E1 -14461.902,E2 -14461.902} C_VEL
LIN {X 0,Y 345.414,Z 698.623,A -85,B 0,C 180,E1 -14462.773,E2 -14462.773} C_VEL
LIN {X 0,Y 347.598,Z 713.262,A -85,B 0,C 180,E1 -14463.267,E2 -14463.267} C_VEL
LIN {X 0,Y 345.458,Z 804.428,A -85,B 0,C 180,E1 -14465.151,E2 -14465.151} C_VEL
LIN {X 0,Y 344.685,Z 818.657,A -85,B 0,C 180,E1 -14465.613,E2 -14465.613} C_VEL
LIN {X 0,Y 343.536,Z 833.127,A -85,B 0,C 180,E1 -14466.329,E2 -14466.329} C_VEL
LIN {X 0,Y 342.258,Z 846.043,A -85,B 0,C 180,E1 -14467.208,E2 -14467.208} C_VEL
LIN {X 0,Y 340.732,Z 859.157,A -85,B 0,C 180,E1 -14468.365,E2 -14468.365} C_VEL
LIN {X 0,Y 339.157,Z 871.137,A -85,B 0,C 180,E1 -14469.69,E2 -14469.69} C_VEL
LIN {X 0,Y 337.518,Z 882.07,A -85,B 0,C 180,E1 -14471.171,E2 -14471.171} C_VEL
LIN {X 0,Y 335.999,Z 892.885,A -85,B 0,C 180,E1 -14472.972,E2 -14472.972} C_VEL
LIN {X 0,Y 334.722,Z 901.951,A -85,B 0,C 180,E1 -14474.816,E2 -14474.816} C_VEL
LIN {X 0,Y 333.802,Z 909.233,A -85,B 0,C 180,E1 -14476.609,E2 -14476.609} C_VEL
LIN {X 0,Y 333.041,Z 915.411,A -85,B 0,C 180,E1 -14478.435,E2 -14478.435} C_VEL
LIN {X 0,Y 332.416,Z 921.977,A -85,B 0,C 180,E1 -14480.876,E2 -14480.876} C_VEL
LIN {X 0,Y 332.115,Z 926.878,A -85,B 0,C 180,E1 -14483.316,E2 -14483.316} C_VEL
LIN {X 0,Y 332.004,Z 929.531,A -85,B 0,C 180,E1 -14485.143,E2 -14485.143} C_VEL
LIN {X 0,Y 331.95,Z 931.839,A -85,B 0,C 180,E1 -14487.573,E2 -14487.573} C_VEL
LIN {X 0,Y 332.043,Z 932.786,A -85,B 0,C 180,E1 -14490,E2 -14490} C_VEL
LIN {X 0,Y 331.936,Z 932.381,A -85,B 0,C 180,E1 -14492.427,E2 -14492.427} C_VEL
LIN {X 0,Y 332.001,Z 930.641,A -85,B 0,C 180,E1 -14494.857,E2 -14494.857} C_VEL
LIN {X 0,Y 332.166,Z 927.525,A -85,B 0,C 180,E1 -14497.293,E2 -14497.293} C_VEL
LIN {X 0,Y 332.566,Z 922.953,A -85,B 0,C 180,E1 -14499.733,E2 -14499.733} C_VEL
LIN {X 0,Y 333.117,Z 918.439,A -85,B 0,C 180,E1 -14501.562,E2 -14501.562} C_VEL
LIN {X 0,Y 334.143,Z 911.957,A -85,B 0,C 180,E1 -14503.687,E2 -14503.687} C_VEL
LIN {X 0,Y 335.288,Z 905.009,A -85,B 0,C 180,E1 -14505.541,E2 -14505.541} C_VEL
LIN {X 0,Y 336.596,Z 897.039,A -85,B 0,C 180,E1 -14507.309,E2 -14507.309} C_VEL
LIN {X 0,Y 338.329,Z 887.269,A -85,B 0,C 180,E1 -14509.097,E2 -14509.097} C_VEL
LIN {X 0,Y 340.239,Z 876.445,A -85,B 0,C 180,E1 -14510.716,E2 -14510.716} C_VEL
LIN {X 0,Y 342.155,Z 864.794,A -85,B 0,C 180,E1 -14512.135,E2 -14512.135} C_VEL
LIN {X 0,Y 343.873,Z 852.7,A -85,B 0,C 180,E1 -14513.327,E2 -14513.327} C_VEL
LIN {X 0,Y 345.513,Z 839.845,A -85,B 0,C 180,E1 -14514.324,E2 -14514.324} C_VEL
LIN {X 0,Y 346.873,Z 826.71,A -85,B 0,C 180,E1 -14515.101,E2 -14515.101} C_VEL
LIN {X 0,Y 348.052,Z 812.478,A -85,B 0,C 180,E1 -14515.69,E2 -14515.69} C_VEL
LIN {X 0,Y 348.732,Z 797.501,A -85,B 0,C 180,E1 -14516.078,E2 -14516.078} C_VEL
LIN {X 0,Y 350.888,Z 712.951,A -85,B 0,C 180,E1 -14517.824,E2 -14517.824} C_VEL
LIN {X 0,Y 346.624,Z 688.896,A -85,B 0,C 180,E1 -14518.79,E2 -14518.79} C_VEL
LIN {X 0,Y 344.371,Z 678.623,A -85,B 0,C 180,E1 -14519.255,E2 -14519.255} C_VEL
LIN {X 0,Y 340.007,Z 668.296,A -85,B 0,C 180,E1 -14519.986,E2 -14519.986} C_VEL
LIN {X 0,Y 336.983,Z 655.513,A -85,B 0,C 180,E1 -14523.465,E2 -14523.465} C_VEL
LIN {X 0,Y 334.402,Z 645.599,A -85,B 0,C 180,E1 -14526.337,E2 -14526.337} C_VEL
LIN {X 0,Y 333.65,Z 643.046,A -85,B 0,C 180,E1 -14527.133,E2 -14527.133} C_VEL
LIN {X 0,Y 333.655,Z 643.04,A -85,B 0,C 180,E1 -14530.766,E2 -14530.766} C_VEL
LIN {X 0,Y 333.618,Z 643.042,A -85,B 0,C 180,E1 -14534.255,E2 -14534.255} C_VEL
LIN {X 0,Y 333.673,Z 643.032,A -85,B 0,C 180,E1 -14537.624,E2 -14537.624} C_VEL
LIN {X 0,Y 333.677,Z 643.039,A -85,B 0,C 180,E1 -14541.197,E2 -14541.197} C_VEL
LIN {X 0,Y 333.686,Z 643.044,A -85,B 0,C 180,E1 -14545.226,E2 -14545.226} C_VEL
LIN {X 0,Y 333.633,Z 643.024,A -85,B 0,C 180,E1 -14548.222,E2 -14548.222} C_VEL
LIN {X 0,Y 333.711,Z 643.036,A -85,B 0,C 180,E1 -14551.028,E2 -14551.028} C_VEL
LIN {X 0,Y 333.736,Z 643.031,A -85,B 0,C 180,E1 -14553.754,E2 -14553.754} C_VEL
LIN {X 0,Y 333.72,Z 643.033,A -85,B 0,C 180,E1 -14557.914,E2 -14557.914} C_VEL
LIN {X 0,Y 333.795,Z 643.024,A -85,B 0,C 180,E1 -14561.59,E2 -14561.59} C_VEL
LIN {X 0,Y 333.809,Z 643.024,A -85,B 0,C 180,E1 -14565.577,E2 -14565.577} C_VEL
LIN {X 0,Y 333.835,Z 643.024,A -85,B 0,C 180,E1 -14569.078,E2 -14569.078} C_VEL
LIN {X 0,Y 334.007,Z 643.004,A -85,B 0,C 180,E1 -14572.747,E2 -14572.747} C_VEL
LIN {X 0,Y 333.81,Z 643.02,A -85,B 0,C 180,E1 -14575.169,E2 -14575.169} C_VEL
LIN {X 0,Y 334.107,Z 642.989,A -85,B 0,C 180,E1 -14577.589,E2 -14577.589} C_VEL
LIN {X 0,Y 334.229,Z 642.97,A -85,B 0,C 180,E1 -14580,E2 -14580} C_VEL
LIN {X 0,Y 334.107,Z 642.991,A -85,B 0,C 180,E1 -14582.412,E2 -14582.412} C_VEL
LIN {X 0,Y 333.993,Z 642.997,A -85,B 0,C 180,E1 -14586.598,E2 -14586.598} C_VEL
LIN {X 0,Y 333.852,Z 643.018,A -85,B 0,C 180,E1 -14589.696,E2 -14589.696} C_VEL
LIN {X 0,Y 333.798,Z 643.028,A -85,B 0,C 180,E1 -14593.392,E2 -14593.392} C_VEL
LIN {X 0,Y 333.749,Z 643.037,A -85,B 0,C 180,E1 -14597.146,E2 -14597.146} C_VEL
LIN {X 0,Y 333.735,Z 643.03,A -85,B 0,C 180,E1 -14599.691,E2 -14599.691} C_VEL
LIN {X 0,Y 333.669,Z 643.038,A -85,B 0,C 180,E1 -14603.591,E2 -14603.591} C_VEL
LIN {X 0,Y 333.665,Z 643.047,A -85,B 0,C 180,E1 -14606.253,E2 -14606.253} C_VEL
LIN {X 0,Y 333.663,Z 643.029,A -85,B 0,C 180,E1 -14610.278,E2 -14610.278} C_VEL
LIN {X 0,Y 333.639,Z 643.047,A -85,B 0,C 180,E1 -14613.209,E2 -14613.209} C_VEL
LIN {X 0,Y 333.677,Z 643.044,A -85,B 0,C 180,E1 -14616.139,E2 -14616.139} C_VEL
LIN {X 0,Y 333.622,Z 643.048,A -85,B 0,C 180,E1 -14619.197,E2 -14619.197} C_VEL
LIN {X 0,Y 333.631,Z 643.05,A -85,B 0,C 180,E1 -14622.5,E2 -14622.5} C_VEL
LIN {X 0,Y 333.596,Z 643.048,A -85,B 0,C 180,E1 -14625.955,E2 -14625.955} C_VEL
LIN {X 0,Y 333.604,Z 643.06,A -85,B 0,C 180,E1 -14629.325,E2 -14629.325} C_VEL
LIN {X 0,Y 333.677,Z 643.132,A -85,B 0,C 180,E1 -14633.248,E2 -14633.248} C_VEL
LIN {X 0,Y 334.767,Z 647.158,A -85,B 0,C 180,E1 -14634.547,E2 -14634.547} C_VEL
LIN {X 0,Y 343.835,Z 665.387,A -85,B 0,C 180,E1 -14635.953,E2 -14635.953} C_VEL
LIN {X 0,Y 351.021,Z 681.586,A -85,B 0,C 180,E1 -14637.041,E2 -14637.041} C_VEL
LIN {X 0,Y 351.589,Z 683.019,A -85,B 0,C 180,E1 -14637.129,E2 -14637.129} C_VEL
LIN {X 0,Y 348.967,Z 783.087,A -85,B 0,C 180,E1 -14639.225,E2 -14639.225} C_VEL
LIN {X 0,Y 348.07,Z 797.555,A -85,B 0,C 180,E1 -14639.752,E2 -14639.752} C_VEL
LIN {X 0,Y 346.779,Z 811.86,A -85,B 0,C 180,E1 -14640.522,E2 -14640.522} C_VEL
LIN {X 0,Y 345.506,Z 823.428,A -85,B 0,C 180,E1 -14641.35,E2 -14641.35} C_VEL
LIN {X 0,Y 343.924,Z 835.696,A -85,B 0,C 180,E1 -14642.462,E2 -14642.462} C_VEL
LIN {X 0,Y 342.12,Z 847.477,A -85,B 0,C 180,E1 -14643.79,E2 -14643.79} C_VEL
LIN {X 0,Y 340.352,Z 858.742,A -85,B 0,C 180,E1 -14645.367,E2 -14645.367} C_VEL
LIN {X 0,Y 338.547,Z 868.848,A -85,B 0,C 180,E1 -14647.093,E2 -14647.093} C_VEL
LIN {X 0,Y 336.906,Z 877.575,A -85,B 0,C 180,E1 -14648.91,E2 -14648.91} C_VEL
LIN {X 0,Y 335.456,Z 885.914,A -85,B 0,C 180,E1 -14651.051,E2 -14651.051} C_VEL
LIN {X 0,Y 334.349,Z 891.695,A -85,B 0,C 180,E1 -14652.886,E2 -14652.886} C_VEL
LIN {X 0,Y 333.54,Z 896.433,A -85,B 0,C 180,E1 -14654.729,E2 -14654.729} C_VEL
LIN {X 0,Y 332.953,Z 900.258,A -85,B 0,C 180,E1 -14656.574,E2 -14656.574} C_VEL
LIN {X 0,Y 332.312,Z 903.976,A -85,B 0,C 180,E1 -14659.028,E2 -14659.028} C_VEL
LIN {X 0,Y 332.123,Z 906.275,A -85,B 0,C 180,E1 -14661.482,E2 -14661.482} C_VEL
LIN {X 0,Y 332.045,Z 907.235,A -85,B 0,C 180,E1 -14663.925,E2 -14663.925} C_VEL
LIN {X 0,Y 332.021,Z 906.884,A -85,B 0,C 180,E1 -14666.359,E2 -14666.359} C_VEL
LIN {X 0,Y 332.083,Z 905.222,A -85,B 0,C 180,E1 -14668.787,E2 -14668.787} C_VEL
LIN {X 0,Y 332.322,Z 902.217,A -85,B 0,C 180,E1 -14671.212,E2 -14671.212} C_VEL
LIN {X 0,Y 332.83,Z 897.784,A -85,B 0,C 180,E1 -14673.632,E2 -14673.632} C_VEL
LIN {X 0,Y 333.459,Z 893.381,A -85,B 0,C 180,E1 -14675.442,E2 -14675.442} C_VEL
LIN {X 0,Y 334.032,Z 888.047,A -85,B 0,C 180,E1 -14677.252,E2 -14677.252} C_VEL
LIN {X 0,Y 335.019,Z 881.612,A -85,B 0,C 180,E1 -14679.052,E2 -14679.052} C_VEL
LIN {X 0,Y 336.046,Z 873.897,A -85,B 0,C 180,E1 -14680.849,E2 -14680.849} C_VEL
LIN {X 0,Y 337.637,Z 864.561,A -85,B 0,C 180,E1 -14682.625,E2 -14682.625} C_VEL
LIN {X 0,Y 339.167,Z 854.246,A -85,B 0,C 180,E1 -14684.245,E2 -14684.245} C_VEL
LIN {X 0,Y 340.684,Z 842.874,A -85,B 0,C 180,E1 -14685.709,E2 -14685.709} C_VEL
LIN {X 0,Y 341.923,Z 831.852,A -85,B 0,C 180,E1 -14686.878,E2 -14686.878} C_VEL
LIN {X 0,Y 343.225,Z 819.991,A -85,B 0,C 180,E1 -14687.887,E2 -14687.887} C_VEL
LIN {X 0,Y 344.363,Z 807.021,A -85,B 0,C 180,E1 -14688.75,E2 -14688.75} C_VEL
LIN {X 0,Y 345.219,Z 793.953,A -85,B 0,C 180,E1 -14689.396,E2 -14689.396} C_VEL
LIN {X 0,Y 345.785,Z 779.844,A -85,B 0,C 180,E1 -14689.865,E2 -14689.865} C_VEL
LIN {X 0,Y 347.855,Z 695.773,A -85,B 0,C 180,E1 -14691.598,E2 -14691.598} C_VEL
LIN {X 0,Y 347.374,Z 691.945,A -85,B 0,C 180,E1 -14691.72,E2 -14691.72} C_VEL
LIN {X 0,Y 346.07,Z 688.356,A -85,B 0,C 180,E1 -14691.902,E2 -14691.902} C_VEL
LIN {X 0,Y 340.044,Z 676.973,A -85,B 0,C 180,E1 -14692.641,E2 -14692.641} C_VEL
LIN {X 0,Y 332.564,Z 658.66,A -85,B 0,C 180,E1 -14693.702,E2 -14693.702} C_VEL
LIN {X 0,Y 327.332,Z 646.911,A -85,B 0,C 180,E1 -14694.459,E2 -14694.459} C_VEL
LIN {X 0,Y 326.606,Z 643.93,A -85,B 0,C 180,E1 -14695.421,E2 -14695.421} C_VEL
LIN {X 0,Y 326.593,Z 643.928,A -85,B 0,C 180,E1 -14698.257,E2 -14698.257} C_VEL
LIN {X 0,Y 326.57,Z 643.933,A -85,B 0,C 180,E1 -14701.098,E2 -14701.098} C_VEL
LIN {X 0,Y 326.609,Z 643.926,A -85,B 0,C 180,E1 -14704.019,E2 -14704.019} C_VEL
LIN {X 0,Y 326.625,Z 643.926,A -85,B 0,C 180,E1 -14707.237,E2 -14707.237} C_VEL
LIN {X 0,Y 326.547,Z 643.926,A -85,B 0,C 180,E1 -14711.124,E2 -14711.124} C_VEL
LIN {X 0,Y 326.562,Z 643.927,A -85,B 0,C 180,E1 -14713.526,E2 -14713.526} C_VEL
LIN {X 0,Y 326.575,Z 643.927,A -85,B 0,C 180,E1 -14717.029,E2 -14717.029} C_VEL
LIN {X 0,Y 326.589,Z 643.918,A -85,B 0,C 180,E1 -14720.778,E2 -14720.778} C_VEL
LIN {X 0,Y 326.613,Z 643.911,A -85,B 0,C 180,E1 -14724.48,E2 -14724.48} C_VEL
LIN {X 0,Y 326.611,Z 643.925,A -85,B 0,C 180,E1 -14727.455,E2 -14727.455} C_VEL
LIN {X 0,Y 326.619,Z 643.913,A -85,B 0,C 180,E1 -14730.336,E2 -14730.336} C_VEL
LIN {X 0,Y 326.644,Z 643.916,A -85,B 0,C 180,E1 -14734.644,E2 -14734.644} C_VEL
LIN {X 0,Y 326.617,Z 643.922,A -85,B 0,C 180,E1 -14738.543,E2 -14738.543} C_VEL
LIN {X 0,Y 326.71,Z 643.905,A -85,B 0,C 180,E1 -14741.175,E2 -14741.175} C_VEL
LIN {X 0,Y 326.766,Z 643.906,A -85,B 0,C 180,E1 -14745.433,E2 -14745.433} C_VEL
LIN {X 0,Y 326.761,Z 643.895,A -85,B 0,C 180,E1 -14748.838,E2 -14748.838} C_VEL
LIN {X 0,Y 326.916,Z 643.885,A -85,B 0,C 180,E1 -14752.589,E2 -14752.589} C_VEL
LIN {X 0,Y 326.765,Z 643.903,A -85,B 0,C 180,E1 -14755.064,E2 -14755.064} C_VEL
LIN {X 0,Y 327.044,Z 643.87,A -85,B 0,C 180,E1 -14757.536,E2 -14757.536} C_VEL
LIN {X 0,Y 327.18,Z 643.849,A -85,B 0,C 180,E1 -14760,E2 -14760} C_VEL
LIN {X 0,Y 327.047,Z 643.87,A -85,B 0,C 180,E1 -14762.463,E2 -14762.463} C_VEL
LIN {X 0,Y 326.984,Z 643.874,A -85,B 0,C 180,E1 -14766.169,E2 -14766.169} C_VEL
LIN {X 0,Y 326.913,Z 643.886,A -85,B 0,C 180,E1 -14768.655,E2 -14768.655} C_VEL
LIN {X 0,Y 326.737,Z 643.909,A -85,B 0,C 180,E1 -14772.421,E2 -14772.421} C_VEL
LIN {X 0,Y 326.756,Z 643.899,A -85,B 0,C 180,E1 -14774.957,E2 -14774.957} C_VEL
LIN {X 0,Y 326.734,Z 643.903,A -85,B 0,C 180,E1 -14778.838,E2 -14778.838} C_VEL
LIN {X 0,Y 326.604,Z 643.92,A -85,B 0,C 180,E1 -14782.788,E2 -14782.788} C_VEL
LIN {X 0,Y 326.691,Z 643.912,A -85,B 0,C 180,E1 -14785.483,E2 -14785.483} C_VEL
LIN {X 0,Y 326.662,Z 643.918,A -85,B 0,C 180,E1 -14789.659,E2 -14789.659} C_VEL
LIN {X 0,Y 326.609,Z 643.924,A -85,B 0,C 180,E1 -14794.019,E2 -14794.019} C_VEL
LIN {X 0,Y 326.631,Z 643.921,A -85,B 0,C 180,E1 -14797.239,E2 -14797.239} C_VEL
LIN {X 0,Y 326.605,Z 643.925,A -85,B 0,C 180,E1 -14800.207,E2 -14800.207} C_VEL
LIN {X 0,Y 326.604,Z 643.924,A -85,B 0,C 180,E1 -14803.518,E2 -14803.518} C_VEL
LIN {X 0,Y 326.583,Z 643.921,A -85,B 0,C 180,E1 -14807.027,E2 -14807.027} C_VEL
LIN {X 0,Y 326.613,Z 643.927,A -85,B 0,C 180,E1 -14810.772,E2 -14810.772} C_VEL
LIN {X 0,Y 326.663,Z 643.95,A -85,B 0,C 180,E1 -14814.439,E2 -14814.439} C_VEL
LIN {X 0,Y 329.566,Z 656.152,A -85,B 0,C 180,E1 -14817.783,E2 -14817.783} C_VEL
LIN {X 0,Y 332.292,Z 668.547,A -85,B 0,C 180,E1 -14821.003,E2 -14821.003} C_VEL
LIN {X 0,Y 335.082,Z 676.361,A -85,B 0,C 180,E1 -14821.427,E2 -14821.427} C_VEL
LIN {X 0,Y 339.86,Z 704.995,A -85,B 0,C 180,E1 -14822.482,E2 -14822.482} C_VEL
LIN {X 0,Y 341.134,Z 713.95,A -85,B 0,C 180,E1 -14822.787,E2 -14822.787} C_VEL
LIN {X 0,Y 338.888,Z 805.526,A -85,B 0,C 180,E1 -14824.717,E2 -14824.717} C_VEL
LIN {X 0,Y 338.018,Z 820.087,A -85,B 0,C 180,E1 -14825.223,E2 -14825.223} C_VEL
LIN {X 0,Y 336.814,Z 834.532,A -85,B 0,C 180,E1 -14825.99,E2 -14825.99} C_VEL
LIN {X 0,Y 335.456,Z 847.29,A -85,B 0,C 180,E1 -14826.902,E2 -14826.902} C_VEL
LIN {X 0,Y 333.9,Z 859.929,A -85,B 0,C 180,E1 -14828.062,E2 -14828.062} C_VEL
LIN {X 0,Y 332.281,Z 871.725,A -85,B 0,C 180,E1 -14829.413,E2 -14829.413} C_VEL
LIN {X 0,Y 330.749,Z 881.528,A -85,B 0,C 180,E1 -14830.77,E2 -14830.77} C_VEL
LIN {X 0,Y 329.148,Z 892.388,A -85,B 0,C 180,E1 -14832.607,E2 -14832.607} C_VEL
LIN {X 0,Y 327.779,Z 901.623,A -85,B 0,C 180,E1 -14834.517,E2 -14834.517} C_VEL
LIN {X 0,Y 326.859,Z 908.808,A -85,B 0,C 180,E1 -14836.319,E2 -14836.319} C_VEL
LIN {X 0,Y 326.038,Z 915.014,A -85,B 0,C 180,E1 -14838.183,E2 -14838.183} C_VEL
LIN {X 0,Y 325.343,Z 921.606,A -85,B 0,C 180,E1 -14840.676,E2 -14840.676} C_VEL
LIN {X 0,Y 325.045,Z 926.533,A -85,B 0,C 180,E1 -14843.17,E2 -14843.17} C_VEL
LIN {X 0,Y 324.915,Z 929.209,A -85,B 0,C 180,E1 -14845.036,E2 -14845.036} C_VEL
LIN {X 0,Y 324.927,Z 930.549,A -85,B 0,C 180,E1 -14846.279,E2 -14846.279} C_VEL
LIN {X 0,Y 324.896,Z 932.192,A -85,B 0,C 180,E1 -14848.76,E2 -14848.76} C_VEL
LIN {X 0,Y 324.948,Z 932.507,A -85,B 0,C 180,E1 -14850,E2 -14850} C_VEL
LIN {X 0,Y 324.854,Z 932.124,A -85,B 0,C 180,E1 -14852.48,E2 -14852.48} C_VEL
LIN {X 0,Y 324.914,Z 930.404,A -85,B 0,C 180,E1 -14854.963,E2 -14854.963} C_VEL
LIN {X 0,Y 325.078,Z 927.31,A -85,B 0,C 180,E1 -14857.453,E2 -14857.453} C_VEL
LIN {X 0,Y 325.517,Z 922.763,A -85,B 0,C 180,E1 -14859.946,E2 -14859.946} C_VEL
LIN {X 0,Y 326.122,Z 918.272,A -85,B 0,C 180,E1 -14861.813,E2 -14861.813} C_VEL
LIN {X 0,Y 327.193,Z 911.818,A -85,B 0,C 180,E1 -14863.984,E2 -14863.984} C_VEL
LIN {X 0,Y 328.344,Z 905.175,A -85,B 0,C 180,E1 -14865.807,E2 -14865.807} C_VEL
LIN {X 0,Y 329.78,Z 896.966,A -85,B 0,C 180,E1 -14867.679,E2 -14867.679} C_VEL
LIN {X 0,Y 331.602,Z 887.238,A -85,B 0,C 180,E1 -14869.5,E2 -14869.5} C_VEL
LIN {X 0,Y 333.6,Z 876.463,A -85,B 0,C 180,E1 -14871.148,E2 -14871.148} C_VEL
LIN {X 0,Y 335.536,Z 865.178,A -85,B 0,C 180,E1 -14872.557,E2 -14872.557} C_VEL
LIN {X 0,Y 337.369,Z 852.86,A -85,B 0,C 180,E1 -14873.804,E2 -14873.804} C_VEL
LIN {X 0,Y 339.079,Z 840.118,A -85,B 0,C 180,E1 -14874.817,E2 -14874.817} C_VEL
LIN {X 0,Y 340.612,Z 825.805,A -85,B 0,C 180,E1 -14875.677,E2 -14875.677} C_VEL
LIN {X 0,Y 341.844,Z 811.193,A -85,B 0,C 180,E1 -14876.274,E2 -14876.274} C_VEL
LIN {X 0,Y 342.558,Z 793.883,A -85,B 0,C 180,E1 -14876.707,E2 -14876.707} C_VEL
LIN {X 0,Y 344.677,Z 713.839,A -85,B 0,C 180,E1 -14878.39,E2 -14878.39} C_VEL
LIN {X 0,Y 340.616,Z 690.749,A -85,B 0,C 180,E1 -14879.342,E2 -14879.342} C_VEL
LIN {X 0,Y 338.569,Z 681.374,A -85,B 0,C 180,E1 -14879.78,E2 -14879.78} C_VEL
LIN {X 0,Y 332.697,Z 667.958,A -85,B 0,C 180,E1 -14880.778,E2 -14880.778} C_VEL
LIN {X 0,Y 329.689,Z 655.109,A -85,B 0,C 180,E1 -14884.395,E2 -14884.395} C_VEL
LIN {X 0,Y 326.615,Z 643.925,A -85,B 0,C 180,E1 -14887.819,E2 -14887.819} C_VEL
LIN {X 0,Y 326.591,Z 643.921,A -85,B 0,C 180,E1 -14891.134,E2 -14891.134} C_VEL
LIN {X 0,Y 326.549,Z 643.926,A -85,B 0,C 180,E1 -14894.747,E2 -14894.747} C_VEL
LIN {X 0,Y 326.598,Z 643.913,A -85,B 0,C 180,E1 -14898.158,E2 -14898.158} C_VEL
LIN {X 0,Y 326.643,Z 643.911,A -85,B 0,C 180,E1 -14901.394,E2 -14901.394} C_VEL
LIN {X 0,Y 326.62,Z 643.922,A -85,B 0,C 180,E1 -14904.851,E2 -14904.851} C_VEL
LIN {X 0,Y 326.61,Z 643.905,A -85,B 0,C 180,E1 -14907.456,E2 -14907.456} C_VEL
LIN {X 0,Y 326.661,Z 643.907,A -85,B 0,C 180,E1 -14910.341,E2 -14910.341} C_VEL
LIN {X 0,Y 326.69,Z 643.912,A -85,B 0,C 180,E1 -14914.517,E2 -14914.517} C_VEL
LIN {X 0,Y 326.647,Z 643.919,A -85,B 0,C 180,E1 -14918.546,E2 -14918.546} C_VEL
LIN {X 0,Y 326.745,Z 643.904,A -85,B 0,C 180,E1 -14921.178,E2 -14921.178} C_VEL
LIN {X 0,Y 326.764,Z 643.903,A -85,B 0,C 180,E1 -14925.433,E2 -14925.433} C_VEL
LIN {X 0,Y 326.771,Z 643.904,A -85,B 0,C 180,E1 -14928.839,E2 -14928.839} C_VEL
LIN {X 0,Y 326.959,Z 643.883,A -85,B 0,C 180,E1 -14932.59,E2 -14932.59} C_VEL
LIN {X 0,Y 326.777,Z 643.896,A -85,B 0,C 180,E1 -14935.065,E2 -14935.065} C_VEL
LIN {X 0,Y 327.047,Z 643.869,A -85,B 0,C 180,E1 -14937.537,E2 -14937.537} C_VEL
LIN {X 0,Y 327.181,Z 643.848,A -85,B 0,C 180,E1 -14940,E2 -14940} C_VEL
LIN {X 0,Y 327.047,Z 643.871,A -85,B 0,C 180,E1 -14942.464,E2 -14942.464} C_VEL
LIN {X 0,Y 326.963,Z 643.872,A -85,B 0,C 180,E1 -14946.589,E2 -14946.589} C_VEL
LIN {X 0,Y 326.807,Z 643.894,A -85,B 0,C 180,E1 -14949.907,E2 -14949.907} C_VEL
LIN {X 0,Y 326.761,Z 643.904,A -85,B 0,C 180,E1 -14953.686,E2 -14953.686} C_VEL
LIN {X 0,Y 326.701,Z 643.913,A -85,B 0,C 180,E1 -14957.528,E2 -14957.528} C_VEL
LIN {X 0,Y 326.661,Z 643.912,A -85,B 0,C 180,E1 -14960.136,E2 -14960.136} C_VEL
LIN {X 0,Y 326.643,Z 643.914,A -85,B 0,C 180,E1 -14964.13,E2 -14964.13} C_VEL
LIN {X 0,Y 326.623,Z 643.901,A -85,B 0,C 180,E1 -14968.254,E2 -14968.254} C_VEL
LIN {X 0,Y 326.575,Z 643.921,A -85,B 0,C 180,E1 -14971.097,E2 -14971.097} C_VEL
LIN {X 0,Y 326.609,Z 643.919,A -85,B 0,C 180,E1 -14974.02,E2 -14974.02} C_VEL
LIN {X 0,Y 326.625,Z 643.921,A -85,B 0,C 180,E1 -14977.238,E2 -14977.238} C_VEL
LIN {X 0,Y 326.545,Z 643.918,A -85,B 0,C 180,E1 -14981.125,E2 -14981.125} C_VEL
LIN {X 0,Y 326.562,Z 643.935,A -85,B 0,C 180,E1 -14983.526,E2 -14983.526} C_VEL
LIN {X 0,Y 326.575,Z 643.934,A -85,B 0,C 180,E1 -14987.029,E2 -14987.029} C_VEL
LIN {X 0,Y 326.584,Z 643.932,A -85,B 0,C 180,E1 -14991.386,E2 -14991.386} C_VEL
LIN {X 0,Y 326.624,Z 644.04,A -85,B 0,C 180,E1 -14992.598,E2 -14992.598} C_VEL
LIN {X 0,Y 327.55,Z 647.5,A -85,B 0,C 180,E1 -14993.738,E2 -14993.738} C_VEL
LIN {X 0,Y 337.145,Z 666.341,A -85,B 0,C 180,E1 -14995.281,E2 -14995.281} C_VEL
LIN {X 0,Y 344.716,Z 683.121,A -85,B 0,C 180,E1 -14996.465,E2 -14996.465} C_VEL
LIN {X 0,Y 345.407,Z 684.921,A -85,B 0,C 180,E1 -14996.576,E2 -14996.576} C_VEL
LIN {X 0,Y 342.759,Z 782.448,A -85,B 0,C 180,E1 -14998.648,E2 -14998.648} C_VEL
LIN {X 0,Y 341.868,Z 796.801,A -85,B 0,C 180,E1 -14999.159,E2 -14999.159} C_VEL
LIN {X 0,Y 340.621,Z 810.601,A -85,B 0,C 180,E1 -14999.892,E2 -14999.892} C_VEL
LIN {X 0,Y 339.311,Z 822.189,A -85,B 0,C 180,E1 -15000.704,E2 -15000.704} C_VEL
LIN {X 0,Y 337.574,Z 835.363,A -85,B 0,C 180,E1 -15001.899,E2 -15001.899} C_VEL
LIN {X 0,Y 335.931,Z 846.072,A -85,B 0,C 180,E1 -15003.101,E2 -15003.101} C_VEL
LIN {X 0,Y 334.23,Z 856.13,A -85,B 0,C 180,E1 -15004.466,E2 -15004.466} C_VEL
LIN {X 0,Y 332.237,Z 867.14,A -85,B 0,C 180,E1 -15006.302,E2 -15006.302} C_VEL
LIN {X 0,Y 330.475,Z 876.203,A -85,B 0,C 180,E1 -15008.151,E2 -15008.151} C_VEL
LIN {X 0,Y 328.804,Z 884.695,A -85,B 0,C 180,E1 -15010.285,E2 -15010.285} C_VEL
LIN {X 0,Y 327.469,Z 891.776,A -85,B 0,C 180,E1 -15012.515,E2 -15012.515} C_VEL
LIN {X 0,Y 326.592,Z 896.556,A -85,B 0,C 180,E1 -15014.396,E2 -15014.396} C_VEL
LIN {X 0,Y 325.979,Z 900.419,A -85,B 0,C 180,E1 -15016.281,E2 -15016.281} C_VEL
LIN {X 0,Y 325.276,Z 904.173,A -85,B 0,C 180,E1 -15018.787,E2 -15018.787} C_VEL
LIN {X 0,Y 325.039,Z 906.507,A -85,B 0,C 180,E1 -15021.295,E2 -15021.295} C_VEL
LIN {X 0,Y 324.958,Z 907.5,A -85,B 0,C 180,E1 -15023.792,E2 -15023.792} C_VEL
LIN {X 0,Y 324.947,Z 907.182,A -85,B 0,C 180,E1 -15026.28,E2 -15026.28} C_VEL
LIN {X 0,Y 324.985,Z 905.555,A -85,B 0,C 180,E1 -15028.761,E2 -15028.761} C_VEL
LIN {X 0,Y 325.232,Z 902.585,A -85,B 0,C 180,E1 -15031.238,E2 -15031.238} C_VEL
LIN {X 0,Y 325.757,Z 898.189,A -85,B 0,C 180,E1 -15033.711,E2 -15033.711} C_VEL
LIN {X 0,Y 326.422,Z 893.825,A -85,B 0,C 180,E1 -15035.56,E2 -15035.56} C_VEL
LIN {X 0,Y 327.015,Z 888.534,A -85,B 0,C 180,E1 -15037.409,E2 -15037.409} C_VEL
LIN {X 0,Y 328.029,Z 882.211,A -85,B 0,C 180,E1 -15039.23,E2 -15039.23} C_VEL
LIN {X 0,Y 329.099,Z 874.475,A -85,B 0,C 180,E1 -15041.081,E2 -15041.081} C_VEL
LIN {X 0,Y 330.762,Z 865.206,A -85,B 0,C 180,E1 -15042.891,E2 -15042.891} C_VEL
LIN {X 0,Y 332.34,Z 854.968,A -85,B 0,C 180,E1 -15044.544,E2 -15044.544} C_VEL
LIN {X 0,Y 333.917,Z 843.688,A -85,B 0,C 180,E1 -15046.036,E2 -15046.036} C_VEL
LIN {X 0,Y 335.184,Z 832.79,A -85,B 0,C 180,E1 -15047.228,E2 -15047.228} C_VEL
LIN {X 0,Y 336.541,Z 821.096,A -85,B 0,C 180,E1 -15048.255,E2 -15048.255} C_VEL
LIN {X 0,Y 337.724,Z 808.383,A -85,B 0,C 180,E1 -15049.133,E2 -15049.133} C_VEL
LIN {X 0,Y 338.642,Z 794.855,A -85,B 0,C 180,E1 -15049.828,E2 -15049.828} C_VEL
LIN {X 0,Y 339.264,Z 781.137,A -85,B 0,C 180,E1 -15050.303,E2 -15050.303} C_VEL
LIN {X 0,Y 341.804,Z 681.724,A -85,B 0,C 180,E1 -15052.389,E2 -15052.389} C_VEL
LIN {X 0,Y 340.044,Z 676.973,A -85,B 0,C 180,E1 -15052.641,E2 -15052.641} C_VEL
LIN {X 0,Y 337.46,Z 672.038,A -85,B 0,C 180,E1 -15052.969,E2 -15052.969} C_VEL
LIN {X 0,Y 324.785,Z 656.442,A -85,B 0,C 180,E1 -15054.456,E2 -15054.456} C_VEL
LIN {X 0,Y 322.891,Z 653.26,A -85,B 0,C 180,E1 -15054.71,E2 -15054.71} C_VEL
LIN {X 0,Y 320.151,Z 647.162,A -85,B 0,C 180,E1 -15055.137,E2 -15055.137} C_VEL
LIN {X 0,Y 319.538,Z 644.807,A -85,B 0,C 180,E1 -15055.944,E2 -15055.944} C_VEL
LIN {X 0,Y 319.527,Z 644.805,A -85,B 0,C 180,E1 -15058.94,E2 -15058.94} C_VEL
LIN {X 0,Y 319.523,Z 644.81,A -85,B 0,C 180,E1 -15061.863,E2 -15061.863} C_VEL
LIN {X 0,Y 319.581,Z 644.801,A -85,B 0,C 180,E1 -15065.542,E2 -15065.542} C_VEL
LIN {X 0,Y 319.531,Z 644.79,A -85,B 0,C 180,E1 -15069.662,E2 -15069.662} C_VEL
LIN {X 0,Y 319.522,Z 644.804,A -85,B 0,C 180,E1 -15073.46,E2 -15073.46} C_VEL
LIN {X 0,Y 319.553,Z 644.802,A -85,B 0,C 180,E1 -15077.016,E2 -15077.016} C_VEL
LIN {X 0,Y 319.548,Z 644.802,A -85,B 0,C 180,E1 -15080.37,E2 -15080.37} C_VEL
LIN {X 0,Y 319.581,Z 644.787,A -85,B 0,C 180,E1 -15084.457,E2 -15084.457} C_VEL
LIN {X 0,Y 319.527,Z 644.804,A -85,B 0,C 180,E1 -15088.137,E2 -15088.137} C_VEL
LIN {X 0,Y 319.574,Z 644.801,A -85,B 0,C 180,E1 -15091.603,E2 -15091.603} C_VEL
LIN {X 0,Y 319.575,Z 644.79,A -85,B 0,C 180,E1 -15095.301,E2 -15095.301} C_VEL
LIN {X 0,Y 319.568,Z 644.801,A -85,B 0,C 180,E1 -15098.045,E2 -15098.045} C_VEL
LIN {X 0,Y 319.627,Z 644.777,A -85,B 0,C 180,E1 -15102.071,E2 -15102.071} C_VEL
LIN {X 0,Y 319.735,Z 644.781,A -85,B 0,C 180,E1 -15106.007,E2 -15106.007} C_VEL
LIN {X 0,Y 319.738,Z 644.765,A -85,B 0,C 180,E1 -15109.872,E2 -15109.872} C_VEL
LIN {X 0,Y 319.904,Z 644.763,A -85,B 0,C 180,E1 -15113.693,E2 -15113.693} C_VEL
LIN {X 0,Y 319.988,Z 644.748,A -85,B 0,C 180,E1 -15117.482,E2 -15117.482} C_VEL
LIN {X 0,Y 320.132,Z 644.727,A -85,B 0,C 180,E1 -15120,E2 -15120} C_VEL
LIN {X 0,Y 319.991,Z 644.749,A -85,B 0,C 180,E1 -15122.517,E2 -15122.517} C_VEL
LIN {X 0,Y 319.94,Z 644.751,A -85,B 0,C 180,E1 -15126.305,E2 -15126.305} C_VEL
LIN {X 0,Y 319.84,Z 644.767,A -85,B 0,C 180,E1 -15128.848,E2 -15128.848} C_VEL
LIN {X 0,Y 319.684,Z 644.786,A -85,B 0,C 180,E1 -15132.699,E2 -15132.699} C_VEL
LIN {X 0,Y 319.702,Z 644.778,A -85,B 0,C 180,E1 -15135.295,E2 -15135.295} C_VEL
LIN {X 0,Y 319.675,Z 644.782,A -85,B 0,C 180,E1 -15139.255,E2 -15139.255} C_VEL
LIN {X 0,Y 319.562,Z 644.797,A -85,B 0,C 180,E1 -15143.32,E2 -15143.32} C_VEL
LIN {X 0,Y 319.636,Z 644.795,A -85,B 0,C 180,E1 -15146.088,E2 -15146.088} C_VEL
LIN {X 0,Y 319.591,Z 644.799,A -85,B 0,C 180,E1 -15148.933,E2 -15148.933} C_VEL
LIN {X 0,Y 319.535,Z 644.804,A -85,B 0,C 180,E1 -15151.861,E2 -15151.861} C_VEL
LIN {X 0,Y 319.581,Z 644.801,A -85,B 0,C 180,E1 -15155.543,E2 -15155.543} C_VEL
LIN {X 0,Y 319.599,Z 644.799,A -85,B 0,C 180,E1 -15158.004,E2 -15158.004} C_VEL
LIN {X 0,Y 319.573,Z 644.8,A -85,B 0,C 180,E1 -15161.606,E2 -15161.606} C_VEL
LIN {X 0,Y 319.523,Z 644.806,A -85,B 0,C 180,E1 -15165.263,E2 -15165.263} C_VEL
LIN {X 0,Y 319.53,Z 644.808,A -85,B 0,C 180,E1 -15168.712,E2 -15168.712} C_VEL
LIN {X 0,Y 319.579,Z 644.804,A -85,B 0,C 180,E1 -15172.344,E2 -15172.344} C_VEL
LIN {X 0,Y 319.618,Z 644.97,A -85,B 0,C 180,E1 -15173.946,E2 -15173.946} C_VEL
LIN {X 0,Y 322.455,Z 656.813,A -85,B 0,C 180,E1 -15177.288,E2 -15177.288} C_VEL
LIN {X 0,Y 325.044,Z 668.351,A -85,B 0,C 180,E1 -15180.354,E2 -15180.354} C_VEL
LIN {X 0,Y 328.931,Z 678.63,A -85,B 0,C 180,E1 -15180.95,E2 -15180.95} C_VEL
LIN {X 0,Y 333.394,Z 705.711,A -85,B 0,C 180,E1 -15181.973,E2 -15181.973} C_VEL
LIN {X 0,Y 334.699,Z 714.937,A -85,B 0,C 180,E1 -15182.296,E2 -15182.296} C_VEL
LIN {X 0,Y 332.399,Z 805.086,A -85,B 0,C 180,E1 -15184.23,E2 -15184.23} C_VEL
LIN {X 0,Y 331.505,Z 819.726,A -85,B 0,C 180,E1 -15184.744,E2 -15184.744} C_VEL
LIN {X 0,Y 330.295,Z 833.626,A -85,B 0,C 180,E1 -15185.485,E2 -15185.485} C_VEL
LIN {X 0,Y 328.898,Z 846.524,A -85,B 0,C 180,E1 -15186.414,E2 -15186.414} C_VEL
LIN {X 0,Y 327.232,Z 859.56,A -85,B 0,C 180,E1 -15187.626,E2 -15187.626} C_VEL
LIN {X 0,Y 325.412,Z 872.31,A -85,B 0,C 180,E1 -15189.123,E2 -15189.123} C_VEL
LIN {X 0,Y 323.679,Z 882.954,A -85,B 0,C 180,E1 -15190.663,E2 -15190.663} C_VEL
LIN {X 0,Y 322.057,Z 893.533,A -85,B 0,C 180,E1 -15192.539,E2 -15192.539} C_VEL
LIN {X 0,Y 320.698,Z 902.257,A -85,B 0,C 180,E1 -15194.427,E2 -15194.427} C_VEL
LIN {X 0,Y 319.721,Z 909.508,A -85,B 0,C 180,E1 -15196.331,E2 -15196.331} C_VEL
LIN {X 0,Y 318.763,Z 916.447,A -85,B 0,C 180,E1 -15198.555,E2 -15198.555} C_VEL
LIN {X 0,Y 318.286,Z 921.234,A -85,B 0,C 180,E1 -15200.467,E2 -15200.467} C_VEL
LIN {X 0,Y 317.97,Z 926.188,A -85,B 0,C 180,E1 -15203.017,E2 -15203.017} C_VEL
LIN {X 0,Y 317.832,Z 928.886,A -85,B 0,C 180,E1 -15204.925,E2 -15204.925} C_VEL
LIN {X 0,Y 317.788,Z 931.24,A -85,B 0,C 180,E1 -15207.465,E2 -15207.465} C_VEL
LIN {X 0,Y 317.853,Z 932.229,A -85,B 0,C 180,E1 -15210,E2 -15210} C_VEL
LIN {X 0,Y 317.774,Z 931.867,A -85,B 0,C 180,E1 -15212.535,E2 -15212.535} C_VEL
LIN {X 0,Y 317.833,Z 930.168,A -85,B 0,C 180,E1 -15215.074,E2 -15215.074} C_VEL
LIN {X 0,Y 318.004,Z 927.095,A -85,B 0,C 180,E1 -15217.62,E2 -15217.62} C_VEL
LIN {X 0,Y 318.486,Z 922.573,A -85,B 0,C 180,E1 -15220.168,E2 -15220.168} C_VEL
LIN {X 0,Y 319.135,Z 918.107,A -85,B 0,C 180,E1 -15222.076,E2 -15222.076} C_VEL
LIN {X 0,Y 320.275,Z 911.681,A -85,B 0,C 180,E1 -15224.292,E2 -15224.292} C_VEL
LIN {X 0,Y 321.688,Z 903.715,A -85,B 0,C 180,E1 -15226.5,E2 -15226.5} C_VEL
LIN {X 0,Y 323.299,Z 895.408,A -85,B 0,C 180,E1 -15228.373,E2 -15228.373} C_VEL
LIN {X 0,Y 325.197,Z 885.426,A -85,B 0,C 180,E1 -15230.23,E2 -15230.23} C_VEL
LIN {X 0,Y 327.421,Z 874.345,A -85,B 0,C 180,E1 -15231.898,E2 -15231.898} C_VEL
LIN {X 0,Y 329.321,Z 863.253,A -85,B 0,C 180,E1 -15233.266,E2 -15233.266} C_VEL
LIN {X 0,Y 331.336,Z 849.724,A -85,B 0,C 180,E1 -15234.599,E2 -15234.599} C_VEL
LIN {X 0,Y 333.199,Z 836.117,A -85,B 0,C 180,E1 -15235.62,E2 -15235.62} C_VEL
LIN {X 0,Y 334.657,Z 822.585,A -85,B 0,C 180,E1 -15236.378,E2 -15236.378} C_VEL
LIN {X 0,Y 335.751,Z 808.791,A -85,B 0,C 180,E1 -15236.914,E2 -15236.914} C_VEL
LIN {X 0,Y 336.57,Z 786.51,A -85,B 0,C 180,E1 -15237.437,E2 -15237.437} C_VEL
LIN {X 0,Y 338.535,Z 714.812,A -85,B 0,C 180,E1 -15238.971,E2 -15238.971} C_VEL
LIN {X 0,Y 334.454,Z 691.62,A -85,B 0,C 180,E1 -15239.959,E2 -15239.959} C_VEL
LIN {X 0,Y 332.789,Z 684.088,A -85,B 0,C 180,E1 -15240.325,E2 -15240.325} C_VEL
LIN {X 0,Y 326.815,Z 670.892,A -85,B 0,C 180,E1 -15241.323,E2 -15241.323} C_VEL
LIN {X 0,Y 325.418,Z 667.617,A -85,B 0,C 180,E1 -15241.61,E2 -15241.61} C_VEL
LIN {X 0,Y 322.812,Z 656.455,A -85,B 0,C 180,E1 -15244.854,E2 -15244.854} C_VEL
LIN {X 0,Y 319.615,Z 644.796,A -85,B 0,C 180,E1 -15248.554,E2 -15248.554} C_VEL
LIN {X 0,Y 319.578,Z 644.795,A -85,B 0,C 180,E1 -15252.979,E2 -15252.979} C_VEL
LIN {X 0,Y 319.578,Z 644.791,A -85,B 0,C 180,E1 -15257.021,E2 -15257.021} C_VEL
LIN {X 0,Y 319.581,Z 644.801,A -85,B 0,C 180,E1 -15260.376,E2 -15260.376} C_VEL
LIN {X 0,Y 319.56,Z 644.787,A -85,B 0,C 180,E1 -15263.573,E2 -15263.573} C_VEL
LIN {X 0,Y 319.577,Z 644.795,A -85,B 0,C 180,E1 -15266.687,E2 -15266.687} C_VEL
LIN {X 0,Y 319.591,Z 644.776,A -85,B 0,C 180,E1 -15269.617,E2 -15269.617} C_VEL
LIN {X 0,Y 319.609,Z 644.794,A -85,B 0,C 180,E1 -15272.498,E2 -15272.498} C_VEL
LIN {X 0,Y 319.605,Z 644.795,A -85,B 0,C 180,E1 -15275.304,E2 -15275.304} C_VEL
LIN {X 0,Y 319.597,Z 644.792,A -85,B 0,C 180,E1 -15278.048,E2 -15278.048} C_VEL
LIN {X 0,Y 319.69,Z 644.782,A -85,B 0,C 180,E1 -15280.962,E2 -15280.962} C_VEL
LIN {X 0,Y 319.732,Z 644.779,A -85,B 0,C 180,E1 -15285.276,E2 -15285.276} C_VEL
LIN {X 0,Y 319.754,Z 644.775,A -85,B 0,C 180,E1 -15289.873,E2 -15289.873} C_VEL
LIN {X 0,Y 319.913,Z 644.759,A -85,B 0,C 180,E1 -15292.426,E2 -15292.426} C_VEL
LIN {X 0,Y 319.746,Z 644.772,A -85,B 0,C 180,E1 -15294.956,E2 -15294.956} C_VEL
LIN {X 0,Y 319.991,Z 644.748,A -85,B 0,C 180,E1 -15297.483,E2 -15297.483} C_VEL
LIN {X 0,Y 320.133,Z 644.725,A -85,B 0,C 180,E1 -15300,E2 -15300} C_VEL
LIN {X 0,Y 319.991,Z 644.751,A -85,B 0,C 180,E1 -15302.518,E2 -15302.518} C_VEL
LIN {X 0,Y 319.925,Z 644.749,A -85,B 0,C 180,E1 -15306.575,E2 -15306.575} C_VEL
LIN {X 0,Y 319.754,Z 644.771,A -85,B 0,C 180,E1 -15310.128,E2 -15310.128} C_VEL
LIN {X 0,Y 319.732,Z 644.774,A -85,B 0,C 180,E1 -15314.725,E2 -15314.725} C_VEL
LIN {X 0,Y 319.69,Z 644.779,A -85,B 0,C 180,E1 -15319.038,E2 -15319.038} C_VEL
LIN {X 0,Y 319.559,Z 644.796,A -85,B 0,C 180,E1 -15323.321,E2 -15323.321} C_VEL
LIN {X 0,Y 319.576,Z 644.801,A -85,B 0,C 180,E1 -15326.094,E2 -15326.094} C_VEL
LIN {X 0,Y 319.554,Z 644.776,A -85,B 0,C 180,E1 -15328.938,E2 -15328.938} C_VEL
LIN {X 0,Y 319.526,Z 644.807,A -85,B 0,C 180,E1 -15331.863,E2 -15331.863} C_VEL
LIN {X 0,Y 319.582,Z 644.802,A -85,B 0,C 180,E1 -15335.543,E2 -15335.543} C_VEL
LIN {X 0,Y 319.529,Z 644.8,A -85,B 0,C 180,E1 -15339.662,E2 -15339.662} C_VEL
LIN {X 0,Y 319.522,Z 644.812,A -85,B 0,C 180,E1 -15343.461,E2 -15343.461} C_VEL
LIN {X 0,Y 319.553,Z 644.808,A -85,B 0,C 180,E1 -15347.016,E2 -15347.016} C_VEL
LIN {X 0,Y 319.548,Z 644.808,A -85,B 0,C 180,E1 -15351.588,E2 -15351.588} C_VEL
LIN {X 0,Y 319.566,Z 644.88,A -85,B 0,C 180,E1 -15351.891,E2 -15351.891} C_VEL
LIN {X 0,Y 320.375,Z 647.891,A -85,B 0,C 180,E1 -15352.891,E2 -15352.891} C_VEL
LIN {X 0,Y 329.809,Z 665.793,A -85,B 0,C 180,E1 -15354.465,E2 -15354.465} C_VEL
LIN {X 0,Y 338.482,Z 684.808,A -85,B 0,C 180,E1 -15355.873,E2 -15355.873} C_VEL
LIN {X 0,Y 339.31,Z 686.861,A -85,B 0,C 180,E1 -15356.009,E2 -15356.009} C_VEL
LIN {X 0,Y 336.535,Z 783.2,A -85,B 0,C 180,E1 -15358.088,E2 -15358.088} C_VEL
LIN {X 0,Y 335.59,Z 797.331,A -85,B 0,C 180,E1 -15358.605,E2 -15358.605} C_VEL
LIN {X 0,Y 334.318,Z 811.065,A -85,B 0,C 180,E1 -15359.351,E2 -15359.351} C_VEL
LIN {X 0,Y 332.944,Z 822.566,A -85,B 0,C 180,E1 -15360.17,E2 -15360.17} C_VEL
LIN {X 0,Y 331.249,Z 835.035,A -85,B 0,C 180,E1 -15361.313,E2 -15361.313} C_VEL
LIN {X 0,Y 329.525,Z 845.849,A -85,B 0,C 180,E1 -15362.535,E2 -15362.535} C_VEL
LIN {X 0,Y 327.658,Z 856.379,A -85,B 0,C 180,E1 -15363.983,E2 -15363.983} C_VEL
LIN {X 0,Y 325.667,Z 867.07,A -85,B 0,C 180,E1 -15365.794,E2 -15365.794} C_VEL
LIN {X 0,Y 323.794,Z 876.19,A -85,B 0,C 180,E1 -15367.676,E2 -15367.676} C_VEL
LIN {X 0,Y 322.087,Z 884.425,A -85,B 0,C 180,E1 -15369.765,E2 -15369.765} C_VEL
LIN {X 0,Y 320.602,Z 891.859,A -85,B 0,C 180,E1 -15372.128,E2 -15372.128} C_VEL
LIN {X 0,Y 319.4,Z 898.099,A -85,B 0,C 180,E1 -15374.69,E2 -15374.69} C_VEL
LIN {X 0,Y 318.762,Z 901.64,A -85,B 0,C 180,E1 -15376.615,E2 -15376.615} C_VEL
LIN {X 0,Y 318.251,Z 904.371,A -85,B 0,C 180,E1 -15378.536,E2 -15378.536} C_VEL
LIN {X 0,Y 317.975,Z 906.739,A -85,B 0,C 180,E1 -15381.1,E2 -15381.1} C_VEL
LIN {X 0,Y 317.881,Z 907.765,A -85,B 0,C 180,E1 -15383.653,E2 -15383.653} C_VEL
LIN {X 0,Y 317.873,Z 907.48,A -85,B 0,C 180,E1 -15386.197,E2 -15386.197} C_VEL
LIN {X 0,Y 317.888,Z 905.888,A -85,B 0,C 180,E1 -15388.733,E2 -15388.733} C_VEL
LIN {X 0,Y 318.143,Z 902.952,A -85,B 0,C 180,E1 -15391.266,E2 -15391.266} C_VEL
LIN {X 0,Y 318.685,Z 898.593,A -85,B 0,C 180,E1 -15393.794,E2 -15393.794} C_VEL
LIN {X 0,Y 319.664,Z 892.652,A -85,B 0,C 180,E1 -15396.311,E2 -15396.311} C_VEL
LIN {X 0,Y 320.373,Z 887.022,A -85,B 0,C 180,E1 -15398.198,E2 -15398.198} C_VEL
LIN {X 0,Y 321.258,Z 881.228,A -85,B 0,C 180,E1 -15399.823,E2 -15399.823} C_VEL
LIN {X 0,Y 322.448,Z 873.596,A -85,B 0,C 180,E1 -15401.631,E2 -15401.631} C_VEL
LIN {X 0,Y 324.169,Z 864.089,A -85,B 0,C 180,E1 -15403.478,E2 -15403.478} C_VEL
LIN {X 0,Y 325.794,Z 853.574,A -85,B 0,C 180,E1 -15405.163,E2 -15405.163} C_VEL
LIN {X 0,Y 327.444,Z 841.948,A -85,B 0,C 180,E1 -15406.683,E2 -15406.683} C_VEL
LIN {X 0,Y 328.866,Z 830.585,A -85,B 0,C 180,E1 -15407.891,E2 -15407.891} C_VEL
LIN {X 0,Y 330.28,Z 818.258,A -85,B 0,C 180,E1 -15408.936,E2 -15408.936} C_VEL
LIN {X 0,Y 331.459,Z 804.593,A -85,B 0,C 180,E1 -15409.831,E2 -15409.831} C_VEL
LIN {X 0,Y 332.302,Z 791.225,A -85,B 0,C 180,E1 -15410.465,E2 -15410.465} C_VEL
LIN {X 0,Y 332.913,Z 776.461,A -85,B 0,C 180,E1 -15410.91,E2 -15410.91} C_VEL
LIN {X 0,Y 335.354,Z 683.382,A -85,B 0,C 180,E1 -15412.881,E2 -15412.881} C_VEL
LIN {X 0,Y 329.247,Z 667.756,A -85,B 0,C 180,E1 -15413.777,E2 -15413.777} C_VEL
LIN {X 0,Y 322.891,Z 653.26,A -85,B 0,C 180,E1 -15414.71,E2 -15414.71} C_VEL
LIN {X 0,Y 320.725,Z 650.295,A -85,B 0,C 180,E1 -15415.05,E2 -15415.05} C_VEL
LIN {X 0,Y 318.187,Z 648.232,A -85,B 0,C 180,E1 -15415.522,E2 -15415.522} C_VEL
LIN {X 0,Y 314.986,Z 646.549,A -85,B 0,C 180,E1 -15416.304,E2 -15416.304} C_VEL
LIN {X 0,Y 312.988,Z 645.833,A -85,B 0,C 180,E1 -15417.113,E2 -15417.113} C_VEL
LIN {X 0,Y 312.482,Z 645.683,A -85,B 0,C 180,E1 -15417.743,E2 -15417.743} C_VEL
LIN {X 0,Y 312.5,Z 645.685,A -85,B 0,C 180,E1 -15421.283,E2 -15421.283} C_VEL
LIN {X 0,Y 312.509,Z 645.682,A -85,B 0,C 180,E1 -15424.21,E2 -15424.21} C_VEL
LIN {X 0,Y 312.513,Z 645.683,A -85,B 0,C 180,E1 -15427.387,E2 -15427.387} C_VEL
LIN {X 0,Y 312.444,Z 645.677,A -85,B 0,C 180,E1 -15430.717,E2 -15430.717} C_VEL
LIN {X 0,Y 312.453,Z 645.683,A -85,B 0,C 180,E1 -15434.21,E2 -15434.21} C_VEL
LIN {X 0,Y 312.457,Z 645.686,A -85,B 0,C 180,E1 -15437.925,E2 -15437.925} C_VEL
LIN {X 0,Y 312.478,Z 645.662,A -85,B 0,C 180,E1 -15441.924,E2 -15441.924} C_VEL
LIN {X 0,Y 312.533,Z 645.662,A -85,B 0,C 180,E1 -15444.22,E2 -15444.22} C_VEL
LIN {X 0,Y 312.504,Z 645.684,A -85,B 0,C 180,E1 -15447.333,E2 -15447.333} C_VEL
LIN {X 0,Y 312.509,Z 645.676,A -85,B 0,C 180,E1 -15451.291,E2 -15451.291} C_VEL
LIN {X 0,Y 312.549,Z 645.671,A -85,B 0,C 180,E1 -15454.707,E2 -15454.707} C_VEL
LIN {X 0,Y 312.529,Z 645.678,A -85,B 0,C 180,E1 -15458.912,E2 -15458.912} C_VEL
LIN {X 0,Y 312.585,Z 645.657,A -85,B 0,C 180,E1 -15461.653,E2 -15461.653} C_VEL
LIN {X 0,Y 312.689,Z 645.662,A -85,B 0,C 180,E1 -15465.686,E2 -15465.686} C_VEL
LIN {X 0,Y 312.688,Z 645.643,A -85,B 0,C 180,E1 -15469.641,E2 -15469.641} C_VEL
LIN {X 0,Y 312.799,Z 645.645,A -85,B 0,C 180,E1 -15472.252,E2 -15472.252} C_VEL
LIN {X 0,Y 312.702,Z 645.654,A -85,B 0,C 180,E1 -15474.842,E2 -15474.842} C_VEL
LIN {X 0,Y 312.989,Z 645.621,A -85,B 0,C 180,E1 -15478.713,E2 -15478.713} C_VEL
LIN {X 0,Y 312.989,Z 645.613,A -85,B 0,C 180,E1 -15481.286,E2 -15481.286} C_VEL
LIN {X 0,Y 312.712,Z 645.653,A -85,B 0,C 180,E1 -15485.157,E2 -15485.157} C_VEL
LIN {X 0,Y 312.859,Z 645.638,A -85,B 0,C 180,E1 -15487.746,E2 -15487.746} C_VEL
LIN {X 0,Y 312.672,Z 645.655,A -85,B 0,C 180,E1 -15491.671,E2 -15491.671} C_VEL
LIN {X 0,Y 312.702,Z 645.65,A -85,B 0,C 180,E1 -15494.887,E2 -15494.887} C_VEL
LIN {X 0,Y 312.631,Z 645.659,A -85,B 0,C 180,E1 -15499.236,E2 -15499.236} C_VEL
LIN {X 0,Y 312.527,Z 645.674,A -85,B 0,C 180,E1 -15502.78,E2 -15502.78} C_VEL
LIN {X 0,Y 312.604,Z 645.67,A -85,B 0,C 180,E1 -15505.935,E2 -15505.935} C_VEL
LIN {X 0,Y 312.547,Z 645.676,A -85,B 0,C 180,E1 -15509.65,E2 -15509.65} C_VEL
LIN {X 0,Y 312.521,Z 645.679,A -85,B 0,C 180,E1 -15513.689,E2 -15513.689} C_VEL
LIN {X 0,Y 312.542,Z 645.676,A -85,B 0,C 180,E1 -15517.383,E2 -15517.383} C_VEL
LIN {X 0,Y 312.503,Z 645.684,A -85,B 0,C 180,E1 -15520.707,E2 -15520.707} C_VEL
LIN {X 0,Y 312.519,Z 645.679,A -85,B 0,C 180,E1 -15524.197,E2 -15524.197} C_VEL
LIN {X 0,Y 312.486,Z 645.682,A -85,B 0,C 180,E1 -15527.918,E2 -15527.918} C_VEL
LIN {X 0,Y 312.536,Z 645.679,A -85,B 0,C 180,E1 -15531.91,E2 -15531.91} C_VEL
LIN {X 0,Y 312.565,Z 645.822,A -85,B 0,C 180,E1 -15533.379,E2 -15533.379} C_VEL
LIN {X 0,Y 315.557,Z 658.028,A -85,B 0,C 180,E1 -15536.931,E2 -15536.931} C_VEL
LIN {X 0,Y 317.744,Z 667.957,A -85,B 0,C 180,E1 -15539.661,E2 -15539.661} C_VEL
LIN {X 0,Y 322.781,Z 680.747,A -85,B 0,C 180,E1 -15540.45,E2 -15540.45} C_VEL
LIN {X 0,Y 326.623,Z 704.28,A -85,B 0,C 180,E1 -15541.364,E2 -15541.364} C_VEL
LIN {X 0,Y 328.281,Z 716.336,A -85,B 0,C 180,E1 -15541.796,E2 -15541.796} C_VEL
LIN {X 0,Y 325.873,Z 806.081,A -85,B 0,C 180,E1 -15543.761,E2 -15543.761} C_VEL
LIN {X 0,Y 324.941,Z 820.139,A -85,B 0,C 180,E1 -15544.283,E2 -15544.283} C_VEL
LIN {X 0,Y 323.694,Z 833.853,A -85,B 0,C 180,E1 -15545.037,E2 -15545.037} C_VEL
LIN {X 0,Y 322.183,Z 847.177,A -85,B 0,C 180,E1 -15546.028,E2 -15546.028} C_VEL
LIN {X 0,Y 320.586,Z 859.129,A -85,B 0,C 180,E1 -15547.165,E2 -15547.165} C_VEL
LIN {X 0,Y 318.763,Z 871.71,A -85,B 0,C 180,E1 -15548.667,E2 -15548.667} C_VEL
LIN {X 0,Y 316.923,Z 882.405,A -85,B 0,C 180,E1 -15550.234,E2 -15550.234} C_VEL
LIN {X 0,Y 315.229,Z 893.031,A -85,B 0,C 180,E1 -15552.148,E2 -15552.148} C_VEL
LIN {X 0,Y 313.808,Z 901.793,A -85,B 0,C 180,E1 -15554.077,E2 -15554.077} C_VEL
LIN {X 0,Y 312.788,Z 909.079,A -85,B 0,C 180,E1 -15556.022,E2 -15556.022} C_VEL
LIN {X 0,Y 311.76,Z 916.048,A -85,B 0,C 180,E1 -15558.294,E2 -15558.294} C_VEL
LIN {X 0,Y 311.246,Z 920.861,A -85,B 0,C 180,E1 -15560.25,E2 -15560.25} C_VEL
LIN {X 0,Y 310.895,Z 925.84,A -85,B 0,C 180,E1 -15562.858,E2 -15562.858} C_VEL
LIN {X 0,Y 310.752,Z 928.563,A -85,B 0,C 180,E1 -15564.81,E2 -15564.81} C_VEL
LIN {X 0,Y 310.71,Z 930.94,A -85,B 0,C 180,E1 -15567.407,E2 -15567.407} C_VEL
LIN {X 0,Y 310.76,Z 931.95,A -85,B 0,C 180,E1 -15570,E2 -15570} C_VEL
LIN {X 0,Y 310.696,Z 931.61,A -85,B 0,C 180,E1 -15572.593,E2 -15572.593} C_VEL
LIN {X 0,Y 310.755,Z 929.932,A -85,B 0,C 180,E1 -15575.19,E2 -15575.19} C_VEL
LIN {X 0,Y 310.951,Z 926.882,A -85,B 0,C 180,E1 -15577.794,E2 -15577.794} C_VEL
LIN {X 0,Y 311.463,Z 922.383,A -85,B 0,C 180,E1 -15580.4,E2 -15580.4} C_VEL
LIN {X 0,Y 312.16,Z 917.944,A -85,B 0,C 180,E1 -15582.35,E2 -15582.35} C_VEL
LIN {X 0,Y 313.377,Z 911.546,A -85,B 0,C 180,E1 -15584.614,E2 -15584.614} C_VEL
LIN {X 0,Y 314.834,Z 903.61,A -85,B 0,C 180,E1 -15586.87,E2 -15586.87} C_VEL
LIN {X 0,Y 316.512,Z 895.34,A -85,B 0,C 180,E1 -15588.782,E2 -15588.782} C_VEL
LIN {X 0,Y 318.518,Z 885.402,A -85,B 0,C 180,E1 -15590.673,E2 -15590.673} C_VEL
LIN {X 0,Y 320.842,Z 874.374,A -85,B 0,C 180,E1 -15592.371,E2 -15592.371} C_VEL
LIN {X 0,Y 322.954,Z 862.226,A -85,B 0,C 180,E1 -15593.895,E2 -15593.895} C_VEL
LIN {X 0,Y 324.906,Z 849.95,A -85,B 0,C 180,E1 -15595.119,E2 -15595.119} C_VEL
LIN {X 0,Y 326.838,Z 836.482,A -85,B 0,C 180,E1 -15596.156,E2 -15596.156} C_VEL
LIN {X 0,Y 328.429,Z 822.412,A -85,B 0,C 180,E1 -15596.961,E2 -15596.961} C_VEL
LIN {X 0,Y 329.539,Z 808.671,A -85,B 0,C 180,E1 -15597.507,E2 -15597.507} C_VEL
LIN {X 0,Y 330.39,Z 786.933,A -85,B 0,C 180,E1 -15598.027,E2 -15598.027} C_VEL
LIN {X 0,Y 332.374,Z 715.362,A -85,B 0,C 180,E1 -15599.591,E2 -15599.591} C_VEL
LIN {X 0,Y 328.21,Z 691.941,A -85,B 0,C 180,E1 -15600.627,E2 -15600.627} C_VEL
LIN {X 0,Y 327.209,Z 687.183,A -85,B 0,C 180,E1 -15600.86,E2 -15600.86} C_VEL
LIN {X 0,Y 321.116,Z 673.828,A -85,B 0,C 180,E1 -15601.911,E2 -15601.911} C_VEL
LIN {X 0,Y 318.157,Z 667.419,A -85,B 0,C 180,E1 -15602.45,E2 -15602.45} C_VEL
LIN {X 0,Y 315.527,Z 656.458,A -85,B 0,C 180,E1 -15605.763,E2 -15605.763} C_VEL
LIN {X 0,Y 312.552,Z 645.677,A -85,B 0,C 180,E1 -15609.321,E2 -15609.321} C_VEL
LIN {X 0,Y 312.529,Z 645.68,A -85,B 0,C 180,E1 -15612.425,E2 -15612.425} C_VEL
LIN {X 0,Y 312.483,Z 645.685,A -85,B 0,C 180,E1 -15616.03,E2 -15616.03} C_VEL
LIN {X 0,Y 312.5,Z 645.678,A -85,B 0,C 180,E1 -15619.293,E2 -15619.293} C_VEL
LIN {X 0,Y 312.541,Z 645.657,A -85,B 0,C 180,E1 -15622.617,E2 -15622.617} C_VEL
LIN {X 0,Y 312.519,Z 645.677,A -85,B 0,C 180,E1 -15626.311,E2 -15626.311} C_VEL
LIN {X 0,Y 312.545,Z 645.664,A -85,B 0,C 180,E1 -15630.35,E2 -15630.35} C_VEL
LIN {X 0,Y 312.603,Z 645.663,A -85,B 0,C 180,E1 -15634.065,E2 -15634.065} C_VEL
LIN {X 0,Y 312.588,Z 645.664,A -85,B 0,C 180,E1 -15637.529,E2 -15637.529} C_VEL
LIN {X 0,Y 312.639,Z 645.658,A -85,B 0,C 180,E1 -15641.657,E2 -15641.657} C_VEL
LIN {X 0,Y 312.695,Z 645.652,A -85,B 0,C 180,E1 -15645.687,E2 -15645.687} C_VEL
LIN {X 0,Y 312.699,Z 645.657,A -85,B 0,C 180,E1 -15649.642,E2 -15649.642} C_VEL
LIN {X 0,Y 312.854,Z 645.635,A -85,B 0,C 180,E1 -15652.254,E2 -15652.254} C_VEL
LIN {X 0,Y 312.717,Z 645.648,A -85,B 0,C 180,E1 -15654.843,E2 -15654.843} C_VEL
LIN {X 0,Y 312.99,Z 645.621,A -85,B 0,C 180,E1 -15658.714,E2 -15658.714} C_VEL
LIN {X 0,Y 312.99,Z 645.614,A -85,B 0,C 180,E1 -15661.287,E2 -15661.287} C_VEL
LIN {X 0,Y 312.717,Z 645.645,A -85,B 0,C 180,E1 -15665.158,E2 -15665.158} C_VEL
LIN {X 0,Y 312.855,Z 645.638,A -85,B 0,C 180,E1 -15667.747,E2 -15667.747} C_VEL
LIN {X 0,Y 312.671,Z 645.658,A -85,B 0,C 180,E1 -15671.672,E2 -15671.672} C_VEL
LIN {X 0,Y 312.702,Z 645.649,A -85,B 0,C 180,E1 -15674.888,E2 -15674.888} C_VEL
LIN {X 0,Y 312.611,Z 645.66,A -85,B 0,C 180,E1 -15679.226,E2 -15679.226} C_VEL
LIN {X 0,Y 312.526,Z 645.675,A -85,B 0,C 180,E1 -15682.78,E2 -15682.78} C_VEL
LIN {X 0,Y 312.535,Z 645.678,A -85,B 0,C 180,E1 -15685.91,E2 -15685.91} C_VEL
LIN {X 0,Y 312.502,Z 645.656,A -85,B 0,C 180,E1 -15689.655,E2 -15689.655} C_VEL
LIN {X 0,Y 312.521,Z 645.675,A -85,B 0,C 180,E1 -15693.689,E2 -15693.689} C_VEL
LIN {X 0,Y 312.516,Z 645.679,A -85,B 0,C 180,E1 -15697.387,E2 -15697.387} C_VEL
LIN {X 0,Y 312.442,Z 645.673,A -85,B 0,C 180,E1 -15700.717,E2 -15700.717} C_VEL
LIN {X 0,Y 312.452,Z 645.687,A -85,B 0,C 180,E1 -15704.21,E2 -15704.21} C_VEL
LIN {X 0,Y 312.457,Z 645.692,A -85,B 0,C 180,E1 -15707.925,E2 -15707.925} C_VEL
LIN {X 0,Y 312.529,Z 645.81,A -85,B 0,C 180,E1 -15711.172,E2 -15711.172} C_VEL
LIN {X 0,Y 313.114,Z 648.073,A -85,B 0,C 180,E1 -15711.977,E2 -15711.977} C_VEL
LIN {X 0,Y 321.726,Z 664.097,A -85,B 0,C 180,E1 -15713.484,E2 -15713.484} C_VEL
LIN {X 0,Y 329.762,Z 680.719,A -85,B 0,C 180,E1 -15714.838,E2 -15714.838} C_VEL
LIN {X 0,Y 333.207,Z 688.883,A -85,B 0,C 180,E1 -15715.418,E2 -15715.418} C_VEL
LIN {X 0,Y 330.341,Z 783.903,A -85,B 0,C 180,E1 -15717.507,E2 -15717.507} C_VEL
LIN {X 0,Y 329.302,Z 798.638,A -85,B 0,C 180,E1 -15718.07,E2 -15718.07} C_VEL
LIN {X 0,Y 327.913,Z 812.673,A -85,B 0,C 180,E1 -15718.865,E2 -15718.865} C_VEL
LIN {X 0,Y 326.546,Z 823.548,A -85,B 0,C 180,E1 -15719.67,E2 -15719.67} C_VEL
LIN {X 0,Y 324.744,Z 836.15,A -85,B 0,C 180,E1 -15720.861,E2 -15720.861} C_VEL
LIN {X 0,Y 322.947,Z 846.814,A -85,B 0,C 180,E1 -15722.103,E2 -15722.103} C_VEL
LIN {X 0,Y 320.896,Z 857.816,A -85,B 0,C 180,E1 -15723.673,E2 -15723.673} C_VEL
LIN {X 0,Y 318.761,Z 868.638,A -85,B 0,C 180,E1 -15725.582,E2 -15725.582} C_VEL
LIN {X 0,Y 316.833,Z 877.539,A -85,B 0,C 180,E1 -15727.503,E2 -15727.503} C_VEL
LIN {X 0,Y 315.042,Z 885.801,A -85,B 0,C 180,E1 -15729.7,E2 -15729.7} C_VEL
LIN {X 0,Y 313.747,Z 891.943,A -85,B 0,C 180,E1 -15731.724,E2 -15731.724} C_VEL
LIN {X 0,Y 312.451,Z 898.224,A -85,B 0,C 180,E1 -15734.341,E2 -15734.341} C_VEL
LIN {X 0,Y 311.792,Z 901.802,A -85,B 0,C 180,E1 -15736.31,E2 -15736.31} C_VEL
LIN {X 0,Y 311.235,Z 904.569,A -85,B 0,C 180,E1 -15738.274,E2 -15738.274} C_VEL
LIN {X 0,Y 310.894,Z 906.972,A -85,B 0,C 180,E1 -15740.895,E2 -15740.895} C_VEL
LIN {X 0,Y 310.806,Z 908.031,A -85,B 0,C 180,E1 -15743.508,E2 -15743.508} C_VEL
LIN {X 0,Y 310.779,Z 907.779,A -85,B 0,C 180,E1 -15746.11,E2 -15746.11} C_VEL
LIN {X 0,Y 310.794,Z 906.22,A -85,B 0,C 180,E1 -15748.704,E2 -15748.704} C_VEL
LIN {X 0,Y 311.054,Z 903.318,A -85,B 0,C 180,E1 -15751.295,E2 -15751.295} C_VEL
LIN {X 0,Y 311.613,Z 898.995,A -85,B 0,C 180,E1 -15753.88,E2 -15753.88} C_VEL
LIN {X 0,Y 312.622,Z 893.107,A -85,B 0,C 180,E1 -15756.454,E2 -15756.454} C_VEL
LIN {X 0,Y 313.383,Z 887.504,A -85,B 0,C 180,E1 -15758.382,E2 -15758.382} C_VEL
LIN {X 0,Y 314.432,Z 880.776,A -85,B 0,C 180,E1 -15760.301,E2 -15760.301} C_VEL
LIN {X 0,Y 315.838,Z 872.703,A -85,B 0,C 180,E1 -15762.204,E2 -15762.204} C_VEL
LIN {X 0,Y 317.598,Z 862.97,A -85,B 0,C 180,E1 -15764.088,E2 -15764.088} C_VEL
LIN {X 0,Y 319.342,Z 852.171,A -85,B 0,C 180,E1 -15765.804,E2 -15765.804} C_VEL
LIN {X 0,Y 321.032,Z 840.2,A -85,B 0,C 180,E1 -15767.354,E2 -15767.354} C_VEL
LIN {X 0,Y 322.533,Z 828.377,A -85,B 0,C 180,E1 -15768.583,E2 -15768.583} C_VEL
LIN {X 0,Y 324.081,Z 815.345,A -85,B 0,C 180,E1 -15769.642,E2 -15769.642} C_VEL
LIN {X 0,Y 325.236,Z 801.136,A -85,B 0,C 180,E1 -15770.516,E2 -15770.516} C_VEL
LIN {X 0,Y 326.041,Z 786.977,A -85,B 0,C 180,E1 -15771.124,E2 -15771.124} C_VEL
LIN {X 0,Y 326.653,Z 767.855,A -85,B 0,C 180,E1 -15771.607,E2 -15771.607} C_VEL
LIN {X 0,Y 328.923,Z 684.9,A -85,B 0,C 180,E1 -15773.395,E2 -15773.395} C_VEL
LIN {X 0,Y 322.394,Z 668.477,A -85,B 0,C 180,E1 -15774.382,E2 -15774.382} C_VEL
LIN {X 0,Y 314.369,Z 650.595,A -85,B 0,C 180,E1 -15775.604,E2 -15775.604} C_VEL
LIN {X 0,Y 312.903,Z 647.418,A -85,B 0,C 180,E1 -15775.86,E2 -15775.86} C_VEL
LIN {X 0,Y 312.498,Z 645.682,A -85,B 0,C 180,E1 -15776.492,E2 -15776.492} C_VEL
LIN {X 0,Y 312.482,Z 645.683,A -85,B 0,C 180,E1 -15777.743,E2 -15777.743} C_VEL
LIN {X 0,Y 311.838,Z 645.767,A -85,B 0,C 180,E1 -15778.819,E2 -15778.819} C_VEL
LIN {X 0,Y 308.949,Z 646.129,A -85,B 0,C 180,E1 -15780.569,E2 -15780.569} C_VEL
LIN {X 0,Y 306.513,Z 646.431,A -85,B 0,C 180,E1 -15781.989,E2 -15781.989} C_VEL
LIN {X 0,Y 305.516,Z 646.555,A -85,B 0,C 180,E1 -15783.089,E2 -15783.089} C_VEL
LIN {X 0,Y 305.462,Z 646.561,A -85,B 0,C 180,E1 -15783.462,E2 -15783.462} C_VEL
LIN {X 0,Y 305.454,Z 646.561,A -85,B 0,C 180,E1 -15786.743,E2 -15786.743} C_VEL
LIN {X 0,Y 305.412,Z 646.551,A -85,B 0,C 180,E1 -15790.59,E2 -15790.59} C_VEL
LIN {X 0,Y 305.427,Z 646.559,A -85,B 0,C 180,E1 -15793.655,E2 -15793.655} C_VEL
LIN {X 0,Y 305.437,Z 646.56,A -85,B 0,C 180,E1 -15797.418,E2 -15797.418} C_VEL
LIN {X 0,Y 305.45,Z 646.54,A -85,B 0,C 180,E1 -15801.593,E2 -15801.593} C_VEL
LIN {X 0,Y 305.464,Z 646.547,A -85,B 0,C 180,E1 -15804.886,E2 -15804.886} C_VEL
LIN {X 0,Y 305.444,Z 646.558,A -85,B 0,C 180,E1 -15808.358,E2 -15808.358} C_VEL
LIN {X 0,Y 305.478,Z 646.55,A -85,B 0,C 180,E1 -15811.109,E2 -15811.109} C_VEL
LIN {X 0,Y 305.502,Z 646.55,A -85,B 0,C 180,E1 -15814.081,E2 -15814.081} C_VEL
LIN {X 0,Y 305.476,Z 646.546,A -85,B 0,C 180,E1 -15816.976,E2 -15816.976} C_VEL
LIN {X 0,Y 305.545,Z 646.539,A -85,B 0,C 180,E1 -15821.214,E2 -15821.214} C_VEL
LIN {X 0,Y 305.63,Z 646.538,A -85,B 0,C 180,E1 -15825.348,E2 -15825.348} C_VEL
LIN {X 0,Y 305.627,Z 646.522,A -85,B 0,C 180,E1 -15829.399,E2 -15829.399} C_VEL
LIN {X 0,Y 305.75,Z 646.524,A -85,B 0,C 180,E1 -15832.072,E2 -15832.072} C_VEL
LIN {X 0,Y 305.671,Z 646.53,A -85,B 0,C 180,E1 -15834.723,E2 -15834.723} C_VEL
LIN {X 0,Y 305.956,Z 646.497,A -85,B 0,C 180,E1 -15838.683,E2 -15838.683} C_VEL
LIN {X 0,Y 305.956,Z 646.489,A -85,B 0,C 180,E1 -15841.316,E2 -15841.316} C_VEL
LIN {X 0,Y 305.684,Z 646.529,A -85,B 0,C 180,E1 -15845.276,E2 -15845.276} C_VEL
LIN {X 0,Y 305.802,Z 646.519,A -85,B 0,C 180,E1 -15847.926,E2 -15847.926} C_VEL
LIN {X 0,Y 305.606,Z 646.538,A -85,B 0,C 180,E1 -15851.945,E2 -15851.945} C_VEL
LIN {X 0,Y 305.64,Z 646.529,A -85,B 0,C 180,E1 -15855.035,E2 -15855.035} C_VEL
LIN {X 0,Y 305.577,Z 646.538,A -85,B 0,C 180,E1 -15859.444,E2 -15859.444} C_VEL
LIN {X 0,Y 305.487,Z 646.55,A -85,B 0,C 180,E1 -15863.039,E2 -15863.039} C_VEL
LIN {X 0,Y 305.549,Z 646.547,A -85,B 0,C 180,E1 -15866.227,E2 -15866.227} C_VEL
LIN {X 0,Y 305.497,Z 646.554,A -85,B 0,C 180,E1 -15869.05,E2 -15869.05} C_VEL
LIN {X 0,Y 305.446,Z 646.56,A -85,B 0,C 180,E1 -15871.952,E2 -15871.952} C_VEL
LIN {X 0,Y 305.464,Z 646.56,A -85,B 0,C 180,E1 -15875.113,E2 -15875.113} C_VEL
LIN {X 0,Y 305.493,Z 646.557,A -85,B 0,C 180,E1 -15878.539,E2 -15878.539} C_VEL
LIN {X 0,Y 305.497,Z 646.556,A -85,B 0,C 180,E1 -15882.594,E2 -15882.594} C_VEL
LIN {X 0,Y 305.445,Z 646.554,A -85,B 0,C 180,E1 -15886.348,E2 -15886.348} C_VEL
LIN {X 0,Y 305.459,Z 646.561,A -85,B 0,C 180,E1 -15889.892,E2 -15889.892} C_VEL
LIN {X 0,Y 305.548,Z 646.731,A -85,B 0,C 180,E1 -15892.807,E2 -15892.807} C_VEL
LIN {X 0,Y 308.558,Z 658.953,A -85,B 0,C 180,E1 -15896.472,E2 -15896.472} C_VEL
LIN {X 0,Y 310.469,Z 667.73,A -85,B 0,C 180,E1 -15898.939,E2 -15898.939} C_VEL
LIN {X 0,Y 316.687,Z 683.063,A -85,B 0,C 180,E1 -15899.939,E2 -15899.939} C_VEL
LIN {X 0,Y 320.909,Z 709.474,A -85,B 0,C 180,E1 -15900.986,E2 -15900.986} C_VEL
LIN {X 0,Y 321.914,Z 717.094,A -85,B 0,C 180,E1 -15901.262,E2 -15901.262} C_VEL
LIN {X 0,Y 319.434,Z 805.632,A -85,B 0,C 180,E1 -15903.234,E2 -15903.234} C_VEL
LIN {X 0,Y 318.429,Z 819.756,A -85,B 0,C 180,E1 -15903.761,E2 -15903.761} C_VEL
LIN {X 0,Y 317.118,Z 834.072,A -85,B 0,C 180,E1 -15904.571,E2 -15904.571} C_VEL
LIN {X 0,Y 315.643,Z 846.395,A -85,B 0,C 180,E1 -15905.5,E2 -15905.5} C_VEL
LIN {X 0,Y 313.831,Z 859.65,A -85,B 0,C 180,E1 -15906.79,E2 -15906.79} C_VEL
LIN {X 0,Y 312.124,Z 871.101,A -85,B 0,C 180,E1 -15908.19,E2 -15908.19} C_VEL
LIN {X 0,Y 310.171,Z 881.851,A -85,B 0,C 180,E1 -15909.785,E2 -15909.785} C_VEL
LIN {X 0,Y 308.404,Z 892.524,A -85,B 0,C 180,E1 -15911.739,E2 -15911.739} C_VEL
LIN {X 0,Y 306.911,Z 901.326,A -85,B 0,C 180,E1 -15913.709,E2 -15913.709} C_VEL
LIN {X 0,Y 305.869,Z 908.649,A -85,B 0,C 180,E1 -15915.7,E2 -15915.7} C_VEL
LIN {X 0,Y 304.773,Z 915.647,A -85,B 0,C 180,E1 -15918.022,E2 -15918.022} C_VEL
LIN {X 0,Y 304.195,Z 920.487,A -85,B 0,C 180,E1 -15920.021,E2 -15920.021} C_VEL
LIN {X 0,Y 303.808,Z 925.492,A -85,B 0,C 180,E1 -15922.69,E2 -15922.69} C_VEL
LIN {X 0,Y 303.685,Z 928.24,A -85,B 0,C 180,E1 -15924.688,E2 -15924.688} C_VEL
LIN {X 0,Y 303.634,Z 930.639,A -85,B 0,C 180,E1 -15927.347,E2 -15927.347} C_VEL
LIN {X 0,Y 303.669,Z 931.671,A -85,B 0,C 180,E1 -15930,E2 -15930} C_VEL
LIN {X 0,Y 303.62,Z 931.354,A -85,B 0,C 180,E1 -15932.653,E2 -15932.653} C_VEL
LIN {X 0,Y 303.685,Z 929.698,A -85,B 0,C 180,E1 -15935.311,E2 -15935.311} C_VEL
LIN {X 0,Y 303.874,Z 926.669,A -85,B 0,C 180,E1 -15937.976,E2 -15937.976} C_VEL
LIN {X 0,Y 304.431,Z 922.194,A -85,B 0,C 180,E1 -15940.643,E2 -15940.643} C_VEL
LIN {X 0,Y 305.197,Z 917.782,A -85,B 0,C 180,E1 -15942.636,E2 -15942.636} C_VEL
LIN {X 0,Y 306.496,Z 911.413,A -85,B 0,C 180,E1 -15944.949,E2 -15944.949} C_VEL
LIN {X 0,Y 307.987,Z 903.51,A -85,B 0,C 180,E1 -15947.256,E2 -15947.256} C_VEL
LIN {X 0,Y 309.756,Z 895.276,A -85,B 0,C 180,E1 -15949.207,E2 -15949.207} C_VEL
LIN {X 0,Y 311.865,Z 885.38,A -85,B 0,C 180,E1 -15951.135,E2 -15951.135} C_VEL
LIN {X 0,Y 314.264,Z 874.402,A -85,B 0,C 180,E1 -15952.865,E2 -15952.865} C_VEL
LIN {X 0,Y 316.539,Z 862.012,A -85,B 0,C 180,E1 -15954.452,E2 -15954.452} C_VEL
LIN {X 0,Y 318.504,Z 850.175,A -85,B 0,C 180,E1 -15955.66,E2 -15955.66} C_VEL
LIN {X 0,Y 320.508,Z 836.847,A -85,B 0,C 180,E1 -15956.713,E2 -15956.713} C_VEL
LIN {X 0,Y 322.123,Z 823.001,A -85,B 0,C 180,E1 -15957.533,E2 -15957.533} C_VEL
LIN {X 0,Y 323.358,Z 808.552,A -85,B 0,C 180,E1 -15958.123,E2 -15958.123} C_VEL
LIN {X 0,Y 324.24,Z 787.318,A -85,B 0,C 180,E1 -15958.641,E2 -15958.641} C_VEL
LIN {X 0,Y 326.315,Z 716.571,A -85,B 0,C 180,E1 -15960.21,E2 -15960.21} C_VEL
LIN {X 0,Y 321.769,Z 690.628,A -85,B 0,C 180,E1 -15961.393,E2 -15961.393} C_VEL
LIN {X 0,Y 314.915,Z 675.42,A -85,B 0,C 180,E1 -15962.624,E2 -15962.624} C_VEL
LIN {X 0,Y 310.877,Z 667.105,A -85,B 0,C 180,E1 -15963.372,E2 -15963.372} C_VEL
LIN {X 0,Y 308.908,Z 658.876,A -85,B 0,C 180,E1 -15965.937,E2 -15965.937} C_VEL
LIN {X 0,Y 305.946,Z 648.263,A -85,B 0,C 180,E1 -15969.491,E2 -15969.491} C_VEL
LIN {X 0,Y 305.466,Z 646.551,A -85,B 0,C 180,E1 -15970.106,E2 -15970.106} C_VEL
LIN {X 0,Y 305.45,Z 646.549,A -85,B 0,C 180,E1 -15973.651,E2 -15973.651} C_VEL
LIN {X 0,Y 305.488,Z 646.542,A -85,B 0,C 180,E1 -15977.407,E2 -15977.407} C_VEL
LIN {X 0,Y 305.508,Z 646.54,A -85,B 0,C 180,E1 -15981.603,E2 -15981.603} C_VEL
LIN {X 0,Y 305.463,Z 646.558,A -85,B 0,C 180,E1 -15984.887,E2 -15984.887} C_VEL
LIN {X 0,Y 305.452,Z 646.531,A -85,B 0,C 180,E1 -15988.355,E2 -15988.355} C_VEL
LIN {X 0,Y 305.521,Z 646.548,A -85,B 0,C 180,E1 -15991.114,E2 -15991.114} C_VEL
LIN {X 0,Y 305.572,Z 646.539,A -85,B 0,C 180,E1 -15994.088,E2 -15994.088} C_VEL
LIN {X 0,Y 305.501,Z 646.55,A -85,B 0,C 180,E1 -15998.403,E2 -15998.403} C_VEL
LIN {X 0,Y 305.591,Z 646.537,A -85,B 0,C 180,E1 -16001.218,E2 -16001.218} C_VEL
LIN {X 0,Y 305.65,Z 646.533,A -85,B 0,C 180,E1 -16005.349,E2 -16005.349} C_VEL
LIN {X 0,Y 305.637,Z 646.537,A -85,B 0,C 180,E1 -16009.4,E2 -16009.4} C_VEL
LIN {X 0,Y 305.798,Z 646.512,A -85,B 0,C 180,E1 -16012.074,E2 -16012.074} C_VEL
LIN {X 0,Y 305.688,Z 646.525,A -85,B 0,C 180,E1 -16014.724,E2 -16014.724} C_VEL
LIN {X 0,Y 305.957,Z 646.497,A -85,B 0,C 180,E1 -16018.684,E2 -16018.684} C_VEL
LIN {X 0,Y 305.957,Z 646.49,A -85,B 0,C 180,E1 -16021.317,E2 -16021.317} C_VEL
LIN {X 0,Y 305.688,Z 646.52,A -85,B 0,C 180,E1 -16025.277,E2 -16025.277} C_VEL
LIN {X 0,Y 305.798,Z 646.518,A -85,B 0,C 180,E1 -16027.926,E2 -16027.926} C_VEL
LIN {X 0,Y 305.605,Z 646.539,A -85,B 0,C 180,E1 -16031.945,E2 -16031.945} C_VEL
LIN {X 0,Y 305.639,Z 646.528,A -85,B 0,C 180,E1 -16035.035,E2 -16035.035} C_VEL
LIN {X 0,Y 305.581,Z 646.538,A -85,B 0,C 180,E1 -16038.783,E2 -16038.783} C_VEL
LIN {X 0,Y 305.488,Z 646.549,A -85,B 0,C 180,E1 -16043.04,E2 -16043.04} C_VEL
LIN {X 0,Y 305.475,Z 646.559,A -85,B 0,C 180,E1 -16046.199,E2 -16046.199} C_VEL
LIN {X 0,Y 305.46,Z 646.53,A -85,B 0,C 180,E1 -16049.038,E2 -16049.038} C_VEL
LIN {X 0,Y 305.438,Z 646.562,A -85,B 0,C 180,E1 -16051.953,E2 -16051.953} C_VEL
LIN {X 0,Y 305.464,Z 646.56,A -85,B 0,C 180,E1 -16055.114,E2 -16055.114} C_VEL
LIN {X 0,Y 305.436,Z 646.565,A -85,B 0,C 180,E1 -16058.525,E2 -16058.525} C_VEL
LIN {X 0,Y 305.437,Z 646.562,A -85,B 0,C 180,E1 -16062.582,E2 -16062.582} C_VEL
LIN {X 0,Y 305.423,Z 646.559,A -85,B 0,C 180,E1 -16066.344,E2 -16066.344} C_VEL
LIN {X 0,Y 305.444,Z 646.763,A -85,B 0,C 180,E1 -16070.415,E2 -16070.415} C_VEL
LIN {X 0,Y 305.961,Z 648.462,A -85,B 0,C 180,E1 -16071.029,E2 -16071.029} C_VEL
LIN {X 0,Y 316.414,Z 667.664,A -85,B 0,C 180,E1 -16072.931,E2 -16072.931} C_VEL
LIN {X 0,Y 324.462,Z 684.497,A -85,B 0,C 180,E1 -16074.337,E2 -16074.337} C_VEL
LIN {X 0,Y 327.128,Z 690.701,A -85,B 0,C 180,E1 -16074.799,E2 -16074.799} C_VEL
